# B&R Automation Studio project NAINV104C00R8L515F00 (part 31)

#### Act_Main.st
```iecst
(** 2019-04-08 **)
ACTION Act_Main:

	IF eStatOld <> eStat THEN
		fbFileOldDel1(bEn := FALSE);
		fbFileRead1(bEn := FALSE);
		fbFileWrite1(bEn := FALSE);

		sStatTxt	:= a_sStatText[eStat];

		eStatOld	:= eStat;

		eStatus		:= Busy;
	END_IF

	//Main
	CASE eStat OF

		HermesActIdle:
			eStatus	:= Idle;

		HermesActBGStartRun:
			IF eStatus = Idle OR eStatus = Busy THEN

				bRun	:= TRUE;
				bStop	:= FALSE;
				eStatus	:= Done;

			END_IF

		HermesActBGStopRun:
			IF eStatus = Idle OR eStatus = Busy THEN

				bStop	:= TRUE;
				eStatus	:= Done;

			END_IF

		HermesActDeleteOldLog:
			IF eStatus = Idle OR eStatus = Busy THEN

				eStatus	:= Busy;

				fbFileOldDel1.dtDTNow	:= p_dtCurrDT;
				fbFileOldDel1(bEn := TRUE);
				IF fbFileOldDel1.udiStatus = 0 THEN
					eStatus	:= Done;
				ELSIF fbFileOldDel1.udiStatus < 65534 THEN
					eStatus		:= Error;

					IF fbFileOldDel1.udiStatus = 1910 THEN
						udiStatus	:= 10111;	//Get Directory Info Error While Deleting Old Log
					ELSIF fbFileOldDel1.udiStatus = 1911 THEN
						udiStatus	:= 10112;	//Directory Read Error While Deleting Old Log
					ELSIF fbFileOldDel1.udiStatus = 1912 THEN
						udiStatus	:= 10113;	//File Delete Error While Deleting Old Log
					ELSE
						udiStatus	:= fbFileOldDel1.udiStatus;
					END_IF
				END_IF

			END_IF
		HermesActReadRetain:
			IF eStatus = Idle OR eStatus = Busy THEN

				eStatus	:= Busy;

				fbFileRead1(bEn := TRUE);

				IF fbFileRead1.udiStatus = 0 THEN
					eStatus	:= Done;

					a_tyBoardDepartedInfoWr := a_tyBoardDepartedInfo;
				ELSIF fbFileRead1.udiStatus < 65534 THEN
					eStatus	:= Error;

					IF fbFileRead1.udiStatus = 1900 THEN
						udiStatus	:= 10114;	//File Open Error While Reading Retain File
					ELSIF fbFileRead1.udiStatus = 1902 THEN
						udiStatus	:= 10115;	//File Read Error While Reading Retain File
					ELSIF fbFileRead1.udiStatus = 1904 THEN
						udiStatus	:= 10116;	//File Close Error While Reading Retain File
					ELSIF fbFileRead1.udiStatus = 1915 THEN
						eStatus			:= Done;
						bFileNotFound	:= TRUE;
					ELSE
						udiStatus	:= fbFileRead1.udiStatus;
					END_IF
				END_IF

			END_IF

		HermesActWriteRetain:
			IF eStatus = Idle OR eStatus = Busy THEN

				eStatus	:= Busy;

				fbFileWrite1(bEn := TRUE);

				IF fbFileWrite1.udiStatus = 0 THEN
					eStatus	:= Done;
				ELSIF fbFileWrite1.udiStatus < 65534 THEN
					eStatus	:= Error;

					IF fbFileWrite1.udiStatus = 1900 THEN
						udiStatus	:= 10117;	//File Open Error While Writing Retain File
					ELSIF fbFileWrite1.udiStatus = 1901 THEN
						udiStatus	:= 10118;	//File Create Error While Writing Retain File
					ELSIF fbFileWrite1.udiStatus = 1903 THEN
						udiStatus	:= 10119;	//File Write Error While Writing Retain File
					ELSIF fbFileWrite1.udiStatus = 1904 THEN
						udiStatus	:= 10120;	//File Close Error While Writing Retain File
					ELSIF fbFileWrite1.udiStatus = 1914 THEN
						udiStatus	:= 10121;	//Directory Does Not Exist While Writing Retain File
					ELSE
						udiStatus	:= fbFileWrite1.udiStatus;
					END_IF
				END_IF

			END_IF

		ELSE
			IF eStatus = Idle OR eStatus = Busy THEN
				eStatus	:= Done;
			END_IF

	END_CASE

END_ACTION
```

#### Init.st
```iecst
(** 2020-09-10 **)
PROGRAM _INIT

	(* Always Change If Project Change *)

	//Pass Address To Global Address For External Use
	//Action, State & Status
	p_DSHermes2Stat		:= ADR(eStat);
	p_DSHermes2Status	:= ADR(eMainStatus);
	p_DSHermes2StatTxt	:= ADR(sStatTxt);

	//Alarm
	p_DSHermes2AlmData	:= ADR(tyAlmData);
	p_DSHermes2AlmData1	:= ADR(tyAlmData1);
	p_DSHermes2AlmData2	:= ADR(tyAlmData2);
	p_DSHermes2AlmData3	:= ADR(tyAlmData3);
	p_DSHermes2AlmData4	:= ADR(tyAlmData4);

	//Output
	p_DSHermes2Connected			:= ADR(bConnected);
	p_DSHermes2HandshakeDone		:= ADR(bHandshakeDone);
	p_DSHermes2USRdy				:= ADR(bUSRdy);
	p_DSHermes2DSRdy				:= ADR(bDSRdy);
	p_DSHermes2USGdRdy				:= ADR(bUSGdRdy);
	p_DSHermes2DSGdRdy				:= ADR(bDSGdRdy);
	p_DSHermes2Transporting			:= ADR(bTransporting);
	p_DSHermes2StopTransport		:= ADR(bStopTransport);
	p_DSHermes2InternalSnd			:= ADR(sInternalSnd);

	p_DSHermes2TransportFinish		:=ADR(bTransportFinishedSnd);
	p_DSHermes2TransportFinishMsg	:= ADR(tyTransportFinished);
	//command
	p_DSHermes2CommandParam			:= ADR(tyCommandParam);
	//route
	p_DSHermes2BrdAvlSnd				:= ADR(tyBoardAvailableSnd);
	//p_DSHermes2RcvReverseUSMcRdy		:= ADR(bDSHermesRcvReverseUSMcRdy);
	(* Always Change If Project Change *)

END_PROGRAM
```

### RmtHermes.var - Change By Project
```iecst
(*2019-05-04*)
(**)
(*Action & State & Status*)
VAR
	p_RmtHermesStat : UDINT;
	p_RmtHermesStatus : UDINT;
	p_RmtHermesStatTxt : UDINT;
	p_RmtHermesAct : UDINT;
	p_RmtHermesMcParamAct : UDINT;
END_VAR
(**)
(*Alarm*)
VAR
	p_RmtHermesAlmData : UDINT;
	p_RmtHermesAlmData1 : UDINT;
	p_RmtHermesAlmData2 : UDINT;
	p_RmtHermesAlmData3 : UDINT;
	p_RmtHermesInfoData : UDINT;
END_VAR
(**)
(*Output*)
VAR
	p_RmtHermesFileNotFound : UDINT;
	p_RmtHermesConnected : UDINT;
	p_RmtHermesWriteConfig : UDINT;
	p_RmtHermesUpdateUIData : UDINT;
	p_RmtHermesSetConfiguration : UDINT;
	p_RmtHermesFoundIndexUS1 : UDINT;
	p_RmtHermesFoundIndexUS2 : UDINT;
	p_RmtHermesFoundIndexUS3 : UDINT;
	p_RmtHermesFoundIndexUS4 : UDINT;
	p_RmtHermesFoundIndexDS1 : UDINT;
	p_RmtHermesFoundIndexDS2 : UDINT;
	p_RmtHermesFoundIndexDS3 : UDINT;
	p_RmtHermesFoundIndexDS4 : UDINT;
	p_RmtHermesIndexUS1 : UDINT;
	p_RmtHermesIndexUS2 : UDINT;
	p_RmtHermesIndexUS3 : UDINT;
	p_RmtHermesIndexUS4 : UDINT;
	p_RmtHermesIndexDS1 : UDINT;
	p_RmtHermesIndexDS2 : UDINT;
	p_RmtHermesIndexDS3 : UDINT;
	p_RmtHermesIndexDS4 : UDINT;
	p_RmtHermesCurrentConfiguration : UDINT;
	p_RmtHermesCurrentConfMcId : UDINT;
END_VAR
```

### Program Logical/Hermes/RmtHermes (IEC, version 1.00.0) - 1.00.0 - NtHermes v5.00.0 , NtTCP v5.00.0 , NtMessage v5.00.0

#### Init.st - Change By Project
```iecst
(** 2021-08-01 **)
PROGRAM _INIT

	(* Always Change If Project Change *)

	//Pass Address To Global Address For External Use
	//Action, State & Status
	p_RmtHermesStat	    	:= ADR(eStat);
	p_RmtHermesStatus   	:= ADR(eMainStatus);
	p_RmtHermesStatTxt   	:= ADR(sStatTxt);
	p_RmtHermesAct	    	:= ADR(eHermesAct);
	p_RmtHermesMcParamAct	:= ADR(eMcParamAct);

	//Alarm
	p_RmtHermesAlmData	    := ADR(tyAlmData);
	p_RmtHermesAlmData1	    := ADR(tyAlmData1);
	p_RmtHermesAlmData2	    := ADR(tyAlmData2);
	p_RmtHermesAlmData3	    := ADR(tyAlmData3);
	p_RmtHermesInfoData	    := ADR(tyInfoData);

	//Output
	p_RmtHermesFileNotFound			:= ADR(bFileNotFound);
	p_RmtHermesConnected			:= ADR(bConnected);
	p_RmtHermesSetConfiguration	    := ADR(tySetConfiguration);
	p_RmtHermesWriteConfig          := ADR(bWriteConfig);
	p_RmtHermesUpdateUIData	        := ADR(bUpdateUIData);

	//Data
	p_RmtHermesFoundIndexUS1              := ADR(bFoundIndexUS1);
	p_RmtHermesFoundIndexUS2              := ADR(bFoundIndexUS2);
	p_RmtHermesFoundIndexUS3              := ADR(bFoundIndexUS3);
	p_RmtHermesFoundIndexUS4              := ADR(bFoundIndexUS4);
	p_RmtHermesFoundIndexDS1              := ADR(bFoundIndexDS1);
	p_RmtHermesFoundIndexDS2              := ADR(bFoundIndexDS2);
	p_RmtHermesFoundIndexDS3              := ADR(bFoundIndexDS3);
	p_RmtHermesFoundIndexDS4              := ADR(bFoundIndexDS4);
	p_RmtHermesIndexUS1                   := ADR(udiFoundIndexUS1);
	p_RmtHermesIndexUS2                   := ADR(udiFoundIndexUS2);
	p_RmtHermesIndexUS3                   := ADR(udiFoundIndexUS3);
	p_RmtHermesIndexUS4                   := ADR(udiFoundIndexUS4);
	p_RmtHermesIndexDS1                   := ADR(udiFoundIndexDS1);
	p_RmtHermesIndexDS2                   := ADR(udiFoundIndexDS2);
	p_RmtHermesIndexDS3                   := ADR(udiFoundIndexDS3);
	p_RmtHermesIndexDS4                   := ADR(udiFoundIndexDS4);
//	p_RmtHermesCurrentConfiguration	:= ADR(tyCurrentConfiguration);
//	p_RmtHermesCurrentConfMcId		:= ADR(tyCurrentConfiguration.tyData.sMachineId);

	(* Always Change If Project Change *)
END_PROGRAM
```

#### Act_InitGlobal.st - Change By Project
```iecst
(** 2021-08-01 **)
ACTION Act_InitGlobal:

	(* Always Change If Project Change *)

	//Pass Data To Link
	p_bLinkStartupRun ACCESS p_StartupRun;

	//Pass Data To Internal Use
	p_udiRstErr ACCESS p_RstErrReset;
	p_bPrep ACCESS p_NtParamHermesPrep;
	p_sIPAddr ACCESS p_HWInfoIPAddr;
	p_tyDTStructure ACCESS p_TimeCurrDTStruct;
	p_dtCurrDT ACCESS p_TimeCurrDT;
	p_sMcId ACCESS p_McParamMcNm;
	p_bRmtPrep ACCESS p_NtParamHermesRmtPrep;
	p_bRmtEn ACCESS p_McParamHermesRmtEn;
	p_udiSndBffrSize ACCESS p_NtParamRmtHermesSndBffrSize;
	p_udiRcvBffrSize ACCESS p_NtParamRmtHermesRcvBffrSize;
	p_udiAliveIdleTimeInSec ACCESS p_NtParamRmtHermesAliveTmInSec;
	p_udiFileKeepDay ACCESS p_NtParamRmtHermesFileKeepDay;
	p_sConfigFileName ACCESS p_NtParamRmtHermesConfigFileNm;
	p_sProgNm ACCESS p_NtParamRmtHermesProgNm;
	p_bNtSettingsLoadDone ACCESS p_StartupNtSettingsLoadDone;
	p_tyHermesConfiguration ACCESS p_HermesConfiguration;
	p_eHermesStat ACCESS p_HermesStat;
	p_eHermesStatus ACCESS p_HermesStatus;
	p_eMcParamStat ACCESS p_McParamStat;
	p_eMcParamStatus ACCESS p_McParamStatus;
	p_iInput ACCESS p_NtParamHermesInput;
	p_iOutput ACCESS p_NtParamHermesOutput;

	(* Always Change If Project Change *)
END_ACTION
```

#### InputRef_Link.var - Change By Project
```iecst
(*2021-08-01*)
(**)
VAR
	p_bLinkStartupRun : REFERENCE TO BOOL;
	bRmtHermesRun : BOOL;
	bRmtHermesStop : BOOL;
END_VAR
```

#### Act_LinkAction.st - Change By Project
```iecst
(** 2021-08-01 **)
ACTION Act_LinkAction:

	IF p_bLinkStartupRun = TRUE THEN
		p_eAct ACCESS p_StartupRmtHermesAct;
	ELSE
		p_eAct ACCESS ADR(eAct);

		IF EDGEPOS(p_bRmtPrep AND p_bRmtEn) THEN
			bRmtHermesRun	:= TRUE;
			bRmtHermesStop	:= FALSE;
		END_IF

		IF EDGENEG(p_bRmtPrep) OR EDGENEG(p_bRmtEn) THEN
			bRmtHermesRun	:= FALSE;
			bRmtHermesStop	:= TRUE;
		END_IF

		IF bRmtHermesRun = TRUE THEN
			p_eAct	:= HermesActBGStartRun;

			IF (eStat = HermesActBGStartRun) AND (eStatus = Done) THEN
				p_eAct			:= HermesActIdle;
				bRmtHermesRun	:= FALSE;
			END_IF
		END_IF

		IF bRmtHermesStop = TRUE THEN
			p_eAct	:= HermesActBGStopRun;

			IF (eStat = HermesActBGStopRun) AND (eStatus = Done) THEN
				p_eAct			:= HermesActIdle;
				bRmtHermesStop	:= FALSE;
			END_IF
		END_IF

	END_IF

END_ACTION
```

#### Act_LinkEn.st - Change By Project
```iecst
(** 2021-08-01 **)
ACTION Act_LinkEn:

	//Link bPrep, bEn & bDis

END_ACTION
```

#### Act_Link.st - Change By Project
```iecst
(** 2021-08-01 **)
ACTION Act_Link:

	//Info Message
	p_sInfoMsg		:= 'Hermes Configuration Received From Remote Station';

	IF	p_iInput > (DINT_TO_INT(c_diHermesConfigMaxIdx)+1) THEN
		p_iInput := (DINT_TO_INT(c_diHermesConfigMaxIdx)+1); //capped at limit
	END_IF

	IF	p_iOutput > (DINT_TO_INT(c_diHermesConfigMaxIdx)+1) THEN
		p_iOutput := (DINT_TO_INT(c_diHermesConfigMaxIdx)+1); //capped at limit
	END_IF

END_ACTION
```

#### Cyclic.st - Do Not Change!!!
```iecst
(** 2021-08-01 **)
PROGRAM _CYCLIC

	IF bInitDone = FALSE THEN
		bInitDone	:= TRUE;

		Act_InitLocal;
		Act_InitGlobal;

	ELSIF bInitialDone = FALSE THEN
		IF p_bNtSettingsLoadDone = TRUE THEN
			bInitialDone	:= TRUE;

			Act_Initial;
		END_IF

	ELSE

		Act_RstErr;
		Act_LinkAction;
		Act_Action;
		Act_LinkEn;

		IF (p_bPrep = TRUE) AND (p_bEn = TRUE) AND (p_bDis = FALSE) THEN
			Act_Link;
			Act_Main;
			Act_Background;
			Act_Background_ProcessData;
		ELSE
			Act_Main_Disable;

			IF eStat <> HermesActIdle THEN
				eStatus	:= Done;
			ELSE
				eStatus	:= Idle;
			END_IF
		END_IF

		Act_CombineErr;
		Act_Alarm;
		Act_Alarm1;
		Act_Alarm2;
		Act_Alarm3;

	END_IF

END_PROGRAM
```

#### Act_RstErr.st - Do Not Change!!!
```iecst
(** 2021-08-01 **)
ACTION Act_RstErr:

	IF p_udiRstErr <> udiRstErrOld THEN
		bRstErr			:= TRUE;
		udiRstErrOld	:= p_udiRstErr;
	ELSE
		bRstErr			:= FALSE;
	END_IF

END_ACTION
```

#### Act_InitLocal.st - Do Not Change!!!
```iecst
(** 2021-08-01 **)
ACTION Act_InitLocal:

	//Input Reference Link To Local Variable
	p_eAct ACCESS ADR(eAct);
	p_udiRstErr ACCESS ADR(udiRstErr);
	p_bPrep ACCESS ADR(bPrep);
	p_bEn ACCESS ADR(bEn);
	p_bDis ACCESS ADR(bDis);
	p_tyParam ACCESS ADR(tyParam);
	p_sIPAddr ACCESS ADR(sIPAddr);
	p_tyDTStructure ACCESS ADR(tyDTStructure);
	p_dtCurrDT ACCESS ADR(dtCurrDT);
	p_sMcId ACCESS ADR(sMcId);
	p_bRmtPrep ACCESS ADR(bRmtPrep);
	p_bRmtEn ACCESS ADR(bRmtEn);
	p_udiSndBffrSize ACCESS ADR(udiSndBffrSize);
	p_udiRcvBffrSize ACCESS ADR(udiRcvBffrSize);
	p_udiAliveIdleTimeInSec ACCESS ADR(udiAliveIdleTimeInSec);
	p_udiFileKeepDay ACCESS ADR(udiFileKeepDay);
	p_sConfigFileName ACCESS ADR(sConfigFileName);
	p_sProgNm ACCESS ADR(sProgNm);
	p_bNtSettingsLoadDone ACCESS ADR(bNtSettingsLoadDone);
	p_sInfoMsg ACCESS ADR(sInfoMsg);
	p_bNtSettingsLoadDone ACCESS ADR(bNtSettingsLoadDone);
	p_sInfoMsg ACCESS ADR(sInfoMsg);
	p_tyHermesConfiguration ACCESS ADR(tyHermesCurrConfiguration);
	p_iInput ACCESS ADR(iInput);
	p_iOutput ACCESS ADR(iOutput);

END_ACTION
```

#### Act_Initial.st - Do Not Change!!!
```iecst
(** 2021-08-01 **)
ACTION Act_Initial:

	//Initial
	sStatTxt	:= a_sStatText[eStat];

	fbCreateSvr.udiSndBffrSize		:= p_udiSndBffrSize;
	fbCreateSvr.udiRcvBffrSize		:= p_udiRcvBffrSize;
	fbCreateSvr.udiAliveIdleTmInSec	:= p_udiAliveIdleTimeInSec;
	fbCreateSvr(bEn := FALSE);

	fbListen(bEn := FALSE);

	fbRcv.udiBffrSize	:= SIZEOF(sRcv);
	fbRcv.p_BffrDest	:= ADR(sRcv);
	fbRcv(bEn := FALSE);

	fbSend.p_BffrDest	:= ADR(sSnd);
	fbSend(bEn := FALSE);

	fbCloseSvr(bEn := FALSE);
	fbCloseClnt(bEn := FALSE);

	fbParseXMLTable.p_XMLTable	:= ADR(a_tyXMLTableDataRcv);

	fbFileAppend1.sDevice	:= 'Log';
	fbFileAppend1(bEn := FALSE);

	fbFileOldDel1.sDevice			:= 'Log';
	fbFileOldDel1.sPath				:= '';
	fbFileOldDel1.sKeyword			:= p_sProgNm;
	fbFileOldDel1.udiFileKeepDay	:= p_udiFileKeepDay;
	fbFileOldDel1(bEn := FALSE);

END_ACTION
```

#### Act_Action.st - Do Not Change!!!
```iecst
(** 2021-08-01 **)
ACTION Act_Action:

	//Reset Error
	IF (eStatus = Error) AND bRstErr THEN
		p_eAct	:= HermesActIdle;
		eStat	:= HermesActIdle;
	END_IF

	//Set p_eAct
	IF eStatus = Idle OR eStatus = Busy OR eStatus = Done THEN
		eStat	:= p_eAct;
	END_IF

END_ACTION
```

#### Act_Main.st - Do Not Change!!!
```iecst
(** 2021-08-01 **)
ACTION Act_Main:

	IF eStatOld <> eStat THEN
		fbFileOldDel1(bEn := FALSE);
		bFileNotFound	:= FALSE;
		sStatTxt	:= a_sStatText[eStat];

		eStatOld	:= eStat;

		eStatus		:= Busy;
	END_IF

	//Main
	CASE eStat OF

		HermesActIdle:
			eStatus	:= Idle;

		HermesActBGStartRun:
			IF eStatus = Idle OR eStatus = Busy THEN

				bRun	:= TRUE;
				bStop	:= FALSE;
				eStatus	:= Done;

			END_IF

		HermesActBGStopRun:
			IF eStatus = Idle OR eStatus = Busy THEN

				bStop	:= TRUE;
				eStatus	:= Done;

			END_IF

		HermesActDeleteOldLog:
			IF eStatus = Idle OR eStatus = Busy THEN

				eStatus	:= Busy;

				fbFileOldDel1.dtDTNow	:= p_dtCurrDT;
				fbFileOldDel1(bEn := TRUE);
				IF fbFileOldDel1.udiStatus = 0 THEN
					eStatus	:= Done;
				ELSIF fbFileOldDel1.udiStatus < 65534 THEN
					eStatus		:= Error;

					IF fbFileOldDel1.udiStatus = 1910 THEN
						udiStatus	:= 10111;	//Get Directory Info Error While Deleting Old Log
					ELSIF fbFileOldDel1.udiStatus = 1911 THEN
						udiStatus	:= 10112;	//Directory Read Error While Deleting Old Log
					ELSIF fbFileOldDel1.udiStatus = 1912 THEN
						udiStatus	:= 10113;	//File Delete Error While Deleting Old Log
					ELSE
						udiStatus	:= fbFileOldDel1.udiStatus;
					END_IF
				END_IF

			END_IF

		ELSE
			IF eStatus = Idle OR eStatus = Busy THEN
				eStatus	:= Done;
			END_IF

	END_CASE

END_ACTION
```

#### Act_Background.st - Do Not Change!!!
```iecst
(** 2021-08-01 **)
ACTION Act_Background:

	IF bRun = TRUE THEN
		IF udiSvrIdent = 0 THEN
			Act_Background_TCPCreateSvr;

			tyParamOld	:= p_tyParam;

		ELSE
			IF bRstConnection = FALSE THEN

				IF udiClntIdent = 0 THEN
					Act_Background_TCPListen;
				END_IF

				IF udiClntIdent <> 0 THEN
					Act_Background_TCPRcv;
				END_IF

				Act_Background_NotificationRcv;

				Act_Background_IllegalMsg;
				Act_Background_UpdtConfig;

				Act_Background_SendConfig;

				Act_Background_Err;

				IF udiClntIdent <> 0 THEN
					Act_Background_TCPSend;
				END_IF

				Act_Background_Log;

			ELSE
				IF udiClntIdent <> 0 THEN
					Act_Background_TCPCloseClnt;
				ELSE
					IF udiSvrIdent <> 0 THEN
						Act_Background_TCPCloseSvr;
					END_IF
				END_IF

			END_IF

		END_IF

		Act_Background_Stop;

	END_IF

	IF EDGENEG(bRun) OR EDGENEG(udiSvrIdent = 0) THEN
		//Reset
		fbCreateSvr(bEn := FALSE);
	END_IF

	IF EDGENEG(bRun) OR EDGENEG(udiClntIdent = 0) THEN
		//Reset
		fbListen(bEn := FALSE);

		bConnected	:= bRun;
	END_IF

	IF EDGENEG(bRun) OR EDGENEG(udiSvrIdent <> 0) OR EDGENEG(udiClntIdent <> 0) THEN
		fbRcv(bEn := FALSE);
		fbSend(bEn := FALSE);

		bConnected		:= FALSE;

		memset(ADR(a_eMsgSend) , 0 , SIZEOF(a_eMsgSend));
		udiMsgSendBffr	:= 0;
	END_IF

	IF EDGENEG(bRun) THEN
		fbFileAppend1(bEn := FALSE);
		iWriteLogStep	:= 0;

		memset(ADR(tyMsgTypeRcv) , 0 , SIZEOF(tyMsgTypeRcv));
	END_IF

	IF EDGENEG(bRun) OR EDGENEG(udiSvrIdent <> 0) THEN
		bRstConnection	:= FALSE;
		fbCloseSvr(bEn := FALSE);
	END_IF

	IF EDGENEG(bRun) OR EDGENEG(udiClntIdent <> 0) THEN
		fbCloseClnt(bEn := FALSE);
	END_IF

	//Reset Error
	IF (eStatus1 = Error) AND bRstErr THEN
		eStatus1	:= Idle;
		udiStatus1	:= 0;

		fbCreateSvr(bEn := FALSE);
		fbListen(bEn := FALSE);
		fbRcv(bEn := FALSE);
		fbSend(bEn := FALSE);
		fbCloseSvr(bEn := FALSE);
		fbCloseClnt(bEn := FALSE);

		fbFileAppend1(bEn := FALSE);
		iWriteLogStep	:= 0;

		bConnected		:= FALSE;
		bRstConnection	:= FALSE;

		memset(ADR(tyMsgTypeRcv) , 0 , SIZEOF(tyMsgTypeRcv));
		memset(ADR(a_eMsgSend) , 0 , SIZEOF(a_eMsgSend));
		udiMsgSendBffr	:= 0;
	END_IF

	IF (eStatus2 = Error) AND bRstErr THEN
		eStatus2	:= Idle;
		udiStatus2	:= 0;

	END_IF

	IF (eStatus3 = Error) AND bRstErr THEN
		eStatus3	:= Idle;
		udiStatus3	:= 0;

		fbFileAppend1(bEn := FALSE);
		iWriteLogStep	:= 0;
	END_IF

END_ACTION
```

#### Act_Background_ProcessData.st - Do Not Change!!!
```iecst
(** 2021-08-01 **)
ACTION Act_Background_ProcessData:

	//Write Config into "Hermes"
	fbDelayTm(IN := bWriteConfig, PT := T#0.5S); //Delay 0.5s to let Hermes take the Data, before WriteConfig

	IF fbDelayTm.Q THEN

		eHermesAct := HermesActWriteConfig;
		eMcParamAct := McParamActWrite;

		IF p_eHermesStatus = Done AND p_eHermesStat = HermesActWriteConfig AND p_eMcParamStat = McParamActWrite AND p_eMcParamStatus = Done THEN

			eMcParamAct     := McParamActIdle;
			eHermesAct		:= HermesActIdle;
			bWriteConfig    := FALSE;
			bUpdateUIData   := TRUE;
			fbDelayTm(IN := FALSE);
			tyInfoData.sProgNm		:= p_sProgNm;
			tyInfoData.udiCode		:= 10000;
			tyInfoData.eSeverity	:= AlmSeverityInfo;
			tyInfoData.sAlmMsg		:= p_sInfoMsg;

		ELSIF  (p_eHermesStatus = Error AND p_eHermesStat = HermesActWriteConfig) OR (p_eMcParamStat = McParamActWrite AND p_eMcParamStatus = Error)  THEN

			eMcParamAct     := McParamActIdle;
			eHermesAct		:= HermesActIdle;
			bWriteConfig    := FALSE;
			bUpdateUIData   := FALSE;
			fbDelayTm(IN := FALSE);

			fHermesAddOneMsgSend(ADR(a_eMsgSend) , ADR(udiMsgSendBffr) , HermesMsgTypeNotification);

			udiStatus2 := 10199; //SetConfiguration Failed, Please Send Again Or Set in Machine HMI back
			tyNotificationSnd.tyAvl.bSeverity			:= TRUE;
			tyNotificationSnd.tyAvl.bNotificationCode	:= TRUE;
			tyNotificationSnd.tyAvl.bDescription		:= TRUE;
			tyNotificationSnd.tyData.eSeverity			:= HermesSeverityFatalError;
			tyNotificationSnd.tyData.iNotificationCode	:= UDINT_TO_INT(udiStatus2);
			tyNotificationSnd.tyData.sDescription		:= a_tyAlmText[udiStatus2].sAlmText;

		END_IF
	END_IF

	//Update UI
	IF bUpdateUIData THEN
		tyInfoData.sProgNm		:= p_sProgNm;
		tyInfoData.udiCode		:= 10000;
		tyInfoData.eSeverity	:= AlmSeverityInfo;
		tyInfoData.sAlmMsg		:= p_sInfoMsg;
	END_IF

	//Auto Reset Info Pop Up
	fbDelayTm1(IN := bUpdateUIData , PT := T#2S); //Auto reset at the Moment (Can Be Changed if need)
	IF fbDelayTm1.Q = TRUE THEN

		//Clear Info Message
		tyInfoData.sProgNm		:= '';
		tyInfoData.udiCode		:= 0;
		tyInfoData.eSeverity	:= AlmSeverityNA;
		tyInfoData.sAlmMsg		:= '';

		bUpdateUIData := FALSE;
		bFoundIndexUS1 := FALSE;
		bFoundIndexUS2 := FALSE;
		bFoundIndexUS3 := FALSE;
		bFoundIndexUS4 := FALSE;
		bFoundIndexDS1 := FALSE;
		bFoundIndexDS2 := FALSE;
		bFoundIndexDS3 := FALSE;
		bFoundIndexDS4 := FALSE;
		fbDelayTm1(IN := FALSE);
	END_IF

END_ACTION
```

#### Act_Background_TCPCreateSvr.st - Do Not Change!!!
```iecst
(** 2021-08-01 **)
ACTION Act_Background_TCPCreateSvr:

	IF eStatus1 <> Error THEN

		//Create Server
		fbCreateSvr.sSvrIP				:= p_sIPAddr;
		fbCreateSvr.uiSvrPort			:= p_tyParam.uiSvrPort; //default = 1248
		fbCreateSvr(bEn := TRUE);

		IF fbCreateSvr.udiStatus = 0 THEN
			udiSvrIdent	:= fbCreateSvr.udiTCPIdent;
			fbCreateSvr(bEn := FALSE);

		ELSIF fbCreateSvr.udiStatus < 65534 THEN
			eStatus1	:= Error;

			IF fbCreateSvr.udiStatus = 2300 THEN
				udiStatus1	:= 10000;	//Invalid Ident While Creating Server
			ELSIF fbCreateSvr.udiStatus = 2302 THEN
				udiStatus1	:= 10001;	//Setting Keep Alive Interval Time Error While Creating Server
			ELSIF fbCreateSvr.udiStatus = 2303 THEN
				udiStatus1	:= 10002;	//Setting Keep Alive Idle Time Error While Creating Server
			ELSIF fbCreateSvr.udiStatus = 2304 THEN
				udiStatus1	:= 10003;	//Setting Keep Alive Count Error While Creating Server
			ELSIF fbCreateSvr.udiStatus = 2305 THEN
				udiStatus1	:= 10004;	//Setting Keep Alive Error While Creating Server
			ELSIF fbCreateSvr.udiStatus = 2306 THEN
				udiStatus1	:= 10005;	//Setting Receive Buffer Error While Creating Server
			ELSIF fbCreateSvr.udiStatus = 2307 THEN
				udiStatus1	:= 10006;	//Setting Send Buffer Error While Creating Server
			ELSIF fbCreateSvr.udiStatus = 2308 THEN
				udiStatus1	:= 10007;	//Setting No Waiting Error While Creating Server
			ELSIF fbCreateSvr.udiStatus = 2309 THEN
				udiStatus1	:= 10008;	//TCP Open Port Error While Creating Server
			ELSIF fbCreateSvr.udiStatus = 2310 THEN
				udiStatus1	:= 10009;	//Closing TCP Error While Creating Server
			ELSE
				udiStatus1	:= fbCreateSvr.udiStatus;
			END_IF

		END_IF

	END_IF

END_ACTION
```

#### Act_Background_TCPListen.st - Do Not Change!!!
```iecst
(** 2021-08-01 **)
ACTION Act_Background_TCPListen:

	IF eStatus1 <> Error AND eStatus2 <> Error THEN

		fbListen.udiSvrIdent	:= udiSvrIdent;
		fbListen(bEn := TRUE);

		IF fbListen.udiStatus = 0 THEN
			udiClntIdent	:= fbListen.udiClntIdent;
			fbListen(bEn := FALSE);

		ELSIF fbListen.udiStatus = 2311 THEN
			fbListen(bEn := FALSE);

		ELSIF fbListen.udiStatus < 65534 THEN
			eStatus1	:= Error;

			IF fbListen.udiStatus = 2300 THEN
				udiStatus1	:= 10010;	//Invalid Ident While Listening Client
			ELSIF fbListen.udiStatus = 2312 THEN
				udiStatus1	:= 10012;	//Listen To Client Error While Listening Client
			ELSE
				udiStatus1	:= fbListen.udiStatus;
			END_IF

		END_IF

	END_IF

END_ACTION
```

#### Act_Background_TCPRcv.st - Do Not Change!!!
```iecst
(** 2021-08-01 **)
ACTION Act_Background_TCPRcv:

	IF eStatus1 <> Error THEN

		//Receive Data
		fbRcv.udiTCPIdent	:= udiClntIdent;
		fbRcv(bEn := TRUE);

		IF fbRcv.udiStatus = 0 THEN

			fLogDTConvert(ADR(sDT) , p_dtCurrDT);
			memset(ADR(a_sLogList[udiLogCntr]) , 0 , SIZEOF(a_sLogList[udiLogCntr]));
			memcpy(ADR(a_sLogList[udiLogCntr]) + LEN(a_sLogList[udiLogCntr]) , ADR(sDT) , LEN(sDT));
			memcpy(ADR(a_sLogList[udiLogCntr]) + LEN(a_sLogList[udiLogCntr]) , ADR('$r$n') , LEN('$r$n'));
			memcpy(ADR(a_sLogList[udiLogCntr]) + LEN(a_sLogList[udiLogCntr]) , ADR('RCV_FRM_RMT$r$n') , LEN('RCV_FRM_RMT$r$n'));
			memcpy(ADR(a_sLogList[udiLogCntr]) + LEN(a_sLogList[udiLogCntr]) , ADR(sRcv) , LEN(sRcv));
			memcpy(ADR(a_sLogList[udiLogCntr]) + LEN(a_sLogList[udiLogCntr]) , ADR('$r$n$r$n') , LEN('$r$n$r$n'));

			udiLogCntr	:= udiLogCntr + 1;
			IF udiLogCntr = 11 THEN
				udiLogCntr	:= 1;
			END_IF

			fXMLConvertToTable(ADR(sRcv) , LEN(sRcv) , ADR(a_tyXMLTableDataRcv) , ADR(a_tyXMLTableDataRcv[0].sTitle) , SIZEOF(a_tyXMLTableDataRcv[0].sTitle) , ADR(a_tyXMLTableDataRcv[0].sValue) , SIZEOF(a_tyXMLTableDataRcv[0].sValue) , ADR(a_tyXMLTableDataRcv[0].uiSize) , SIZEOF(a_tyXMLTableDataRcv[0]) , SIZEOF(a_tyXMLTableDataRcv) / SIZEOF(a_tyXMLTableDataRcv[0]) , ADR(udiXMLTableWriteIdx));

			fbParseXMLTable.iTotalIdxWrite	:= UDINT_TO_INT(udiXMLTableWriteIdx);
			fbParseXMLTable;

			IF fbParseXMLTable.tyMsgType.bCheckAlive = TRUE THEN
				tyMsgTypeRcv.bCheckAlive	:= TRUE;
				tyCheckAlive				:= fbParseXMLTable.tyCheckAlive;
			END_IF

			IF fbParseXMLTable.tyMsgType.bCheckAlivePing = TRUE THEN
				tyMsgTypeRcv.bCheckAlivePing	:= TRUE;
				tyCheckAlivePing				:= fbParseXMLTable.tyCheckAlivePing;
			END_IF

			IF fbParseXMLTable.tyMsgType.bCheckAlivePong = TRUE THEN
				tyMsgTypeRcv.bCheckAlivePong	:= TRUE;
				tyCheckAlivePong				:= fbParseXMLTable.tyCheckAlivePong;
			END_IF

			IF fbParseXMLTable.tyMsgType.bServiceDescription = TRUE THEN
				tyMsgTypeRcv.bServiceDescription	:= TRUE;
				tyServiceDescriptionRcv				:= fbParseXMLTable.tyServiceDescription;
			END_IF

			IF fbParseXMLTable.tyMsgType.bNotification = TRUE THEN
				tyMsgTypeRcv.bNotification	:= TRUE;
				tyNotificationRcv			:= fbParseXMLTable.tyNotification;
			END_IF

			IF fbParseXMLTable.tyMsgType.bBoardAvailable = TRUE THEN
				tyMsgTypeRcv.bBoardAvailable	:= TRUE;
				tyBoardAvailableRcv				:= fbParseXMLTable.tyBoardAvailable;

			END_IF

			IF fbParseXMLTable.tyMsgType.bRevokeBoardAvailable = TRUE THEN
				tyMsgTypeRcv.bRevokeBoardAvailable	:= TRUE;
			END_IF

			IF fbParseXMLTable.tyMsgType.bMachineReady = TRUE THEN
				tyMsgTypeRcv.bMachineReady	:= TRUE;
				tyMachineReady				:= fbParseXMLTable.tyMachineReady;
			END_IF

			IF fbParseXMLTable.tyMsgType.bRevokeMachineReady = TRUE THEN
				tyMsgTypeRcv.bRevokeMachineReady	:= TRUE;
			END_IF

			IF fbParseXMLTable.tyMsgType.bStartTransport = TRUE THEN
				tyMsgTypeRcv.bStartTransport	:= TRUE;
				tyStartTransport				:= fbParseXMLTable.tyStartTransport;
			END_IF

			IF fbParseXMLTable.tyMsgType.bStopTransport = TRUE THEN
				tyMsgTypeRcv.bStopTransport	:= TRUE;
				tyStopTransport				:= fbParseXMLTable.tyStopTransport;
			END_IF

			IF fbParseXMLTable.tyMsgType.bTransportFinished = TRUE THEN
				tyMsgTypeRcv.bTransportFinished	:= TRUE;
				tyTransportFinished				:= fbParseXMLTable.tyTransportFinished;
			END_IF

			IF fbParseXMLTable.tyMsgType.bSetConfiguration = TRUE THEN
				tyMsgTypeRcv.bSetConfiguration	:= TRUE;
				tySetConfigurationRcv			:= fbParseXMLTable.tySetConfiguration;
			END_IF

			IF fbParseXMLTable.tyMsgType.bGetConfiguration = TRUE THEN
				tyMsgTypeRcv.bGetConfiguration	:= TRUE;
			END_IF

			IF fbParseXMLTable.tyMsgType.bCurrentConfiguration = TRUE THEN
				tyMsgTypeRcv.bCurrentConfiguration	:= TRUE;
				tyCurrentConfigurationRcv			:= fbParseXMLTable.tyCurrentConfiguration;
			END_IF

			IF fbParseXMLTable.tyMsgType.bBoardForecast = TRUE THEN
				tyMsgTypeRcv.bBoardForecast	:= TRUE;
				tyBoardForecast				:= fbParseXMLTable.tyBoardForecast;
			END_IF

			IF fbParseXMLTable.tyMsgType.bQueryBoardInfo = TRUE THEN
				tyMsgTypeRcv.bQueryBoardInfo	:= TRUE;
				tyQueryBoardInfo				:= fbParseXMLTable.tyQueryBoardInfo;
			END_IF

			IF fbParseXMLTable.tyMsgType.bSendBoardInfo = TRUE THEN
				tyMsgTypeRcv.bSendBoardInfo	:= TRUE;
				tySendBoardInfo				:= fbParseXMLTable.tySendBoardInfo;
			END_IF

			fbRcv(bEn := FALSE);

			memset(ADR(sRcv) , 0 , SIZEOF(sRcv));

		ELSIF fbRcv.udiStatus = 2317 THEN
			fbRcv(bEn := FALSE);

			memset(ADR(sRcv) , 0 , SIZEOF(sRcv));

		ELSIF fbRcv.udiStatus = 2316 THEN
			bRstConnection	:= TRUE;

			memset(ADR(sRcv) , 0 , SIZEOF(sRcv));

		ELSIF fbRcv.udiStatus = 2318 THEN
			bRstConnection	:= TRUE;

			memset(ADR(sRcv) , 0 , SIZEOF(sRcv));

		ELSIF fbRcv.udiStatus < 65534 THEN
			eStatus1	:= Error;

			IF fbRcv.udiStatus = 2300 THEN
				udiStatus1	:= 10014;	//Invalid Ident While Receiving Data
			ELSIF fbRcv.udiStatus = 2319 THEN
				udiStatus1	:= 10015;	//TCP Receive Data Error While Receiving Data
			ELSE
				udiStatus1	:= fbRcv.udiStatus;
			END_IF

			memset(ADR(sRcv) , 0 , SIZEOF(sRcv));

		END_IF

	END_IF

END_ACTION
```

#### Act_Background_NotificationRcv.st - Do Not Change!!!
```iecst
(** 2021-08-01 **)
ACTION Act_Background_NotificationRcv:

	IF eStatus1 <> Error THEN

		IF tyMsgTypeRcv.bNotification = TRUE THEN
			tyMsgTypeRcv.bNotification	:= FALSE;

			bRstConnection	:= fHermesNotificationRstConn(tyNotificationRcv) OR bRstConnection;

		END_IF

	END_IF

END_ACTION
```

#### Act_Background_IllegalMsg.st - Do Not Change!!!
```iecst
(** 2021-08-01 **)
ACTION Act_Background_IllegalMsg:

	IF eStatus2 <> Error THEN

		udiStatus2	:= fHermesIllegalMsgRmt(tyMsgTypeRcv);

		IF udiStatus2 <> 0 THEN
			eStatus2	:= Error;

			IF udiStatus2 = 2925 THEN
				udiStatus2	:= 10114;	//Receive Check Alive While In Remote Configuration
			ELSIF udiStatus2 = 2926 THEN
				udiStatus2	:= 10115;	//Receive Check Alive Ping While In Remote Configuration
			ELSIF udiStatus2 = 2927 THEN
				udiStatus2	:= 10116;	//Receive Check Alive Pong While In Remote Configuration
			ELSIF udiStatus2 = 2928 THEN
				udiStatus2	:= 10117;	//Receive ServiceDescription While In Remote Configuration
			ELSIF udiStatus2 = 2929 THEN
				udiStatus2	:= 10118;	//Receive BoardAvailable While In Remote Configuration
			ELSIF udiStatus2 = 2930 THEN
				udiStatus2	:= 10119;	//Receive RevokeBoardAvailable While In Remote Configuration
			ELSIF udiStatus2 = 2931 THEN
				udiStatus2	:= 10120;	//Receive MachineReady While In Remote Configuration
			ELSIF udiStatus2 = 2932 THEN
				udiStatus2	:= 10121;	//Receive RevokeMachineReady While In Remote Configuration
			ELSIF udiStatus2 = 2933 THEN
				udiStatus2	:= 10122;	//Receive StartTransport While In Remote Configuration
			ELSIF udiStatus2 = 2934 THEN
				udiStatus2	:= 10123;	//Receive StopTransport While In Remote Configuration
			ELSIF udiStatus2 = 2935 THEN
				udiStatus2	:= 10124;	//Receive TransportFinished While In Remote Configuration
			ELSIF udiStatus2 = 2936 THEN
				udiStatus2	:= 10125;	//Receive CurrentConfiguration While In Remote Configuration
			ELSIF udiStatus2 = 2937 THEN
				udiStatus2	:= 10126;	//Receive BoardForecast While In Remote Configuration
			ELSIF udiStatus2 = 2938 THEN
				udiStatus2	:= 10127;	//Receive QueryBoardInfo While In Remote Configuration
			ELSIF udiStatus2 = 2939 THEN
				udiStatus2	:= 10128;	//Receive SendBoardInfo While In Remote Configuration
			END_IF

			fHermesAddOneMsgSend(ADR(a_eMsgSend) , ADR(udiMsgSendBffr) , HermesMsgTypeNotification);

			tyNotificationSnd.tyAvl.bSeverity			:= TRUE;
			tyNotificationSnd.tyAvl.bNotificationCode	:= TRUE;
			tyNotificationSnd.tyAvl.bDescription		:= TRUE;
			tyNotificationSnd.tyData.eSeverity			:= HermesSeverityFatalError;
			tyNotificationSnd.tyData.iNotificationCode	:= UDINT_TO_INT(udiStatus2);
			tyNotificationSnd.tyData.sDescription		:= a_tyAlmText[udiStatus2].sAlmText;

		END_IF

	END_IF

END_ACTION
```

#### Act_Background_ChkParamRcv.st - Do Not Change!!!
```iecst
(** 2019-05-04 **)
ACTION Act_Background_ChkParamRcv:

//	IF eStatus2 <> Error THEN

		//Check Parameter Receive
//		IF tyMsgTypeRcv.bSetConfiguration = TRUE THEN

//				fHermesAddOneMsgSend(ADR(a_eMsgSend) , ADR(udiMsgSendBffr) , HermesMsgTypeNotification);
//
//				tyNotificationSnd.tyAvl.bSeverity			:= TRUE;
//				tyNotificationSnd.tyAvl.bNotificationCode	:= TRUE;
//				tyNotificationSnd.tyAvl.bDescription		:= TRUE;
//				tyNotificationSnd.tyData.eSeverity			:= HermesSeverityFatalError;
//				tyNotificationSnd.tyData.iNotificationCode	:= 4;
//				tyNotificationSnd.tyData.sDescription		:= a_tyAlmText[udiStatus2].sAlmText;

//		END_IF
//	END_IF

END_ACTION
```

#### Act_Background_UpdtConfig.st - Do Not Change!!!
```iecst
(** 2021-08-01 **)
ACTION Act_Background_UpdtConfig:

	IF eStatus2 <> Error THEN

		IF tyMsgTypeRcv.bSetConfiguration = TRUE THEN

			tySetConfiguration.tyAvl.bMachineId						:= tySetConfigurationRcv.tyAvl.bMachineId;
			tySetConfiguration.tyAvl.bSupervisorySystemPort			:= tySetConfigurationRcv.tyAvl.bSupervisorySystemPort;
			tySetConfiguration.tyAvl.bUpstreamConfigurations		:= tySetConfigurationRcv.tyAvl.bUpstreamConfigurations;
			tySetConfiguration.tyAvl.bDownstreamConfigurations		:= tySetConfigurationRcv.tyAvl.bDownstreamConfigurations;
			tySetConfiguration.tyAvl.iUpstreamConfigurations		:= tySetConfigurationRcv.tyAvl.iUpstreamConfigurations;
			tySetConfiguration.tyAvl.iDownstreamConfigurations		:= tySetConfigurationRcv.tyAvl.iDownstreamConfigurations;
			tySetConfiguration.tyAvl.a_tyUpstreamConfigurations		:= tySetConfigurationRcv.tyAvl.a_tyUpstreamConfigurations;
			tySetConfiguration.tyAvl.a_tyDownstreamConfigurations	:= tySetConfigurationRcv.tyAvl.a_tyDownstreamConfigurations;

			tySetConfiguration.tyData.sMachineId					:= tySetConfigurationRcv.tyData.sMachineId;
			tySetConfiguration.tyData.uiSupervisorySystemPort		:= tySetConfigurationRcv.tyData.uiSupervisorySystemPort;
			tySetConfiguration.tyData.a_tyUpstreamConfigurations	:= tySetConfigurationRcv.tyData.a_tyUpstreamConfigurations;
			tySetConfiguration.tyData.a_tyDownstreamConfigurations	:= tySetConfigurationRcv.tyData.a_tyDownstreamConfigurations;

			udiTargetAddress := ADR(tySetConfiguration.tyData.a_tyUpstreamConfigurations[0].iUpstreamLaneId); //Start address
			udiSizeAddress   := SIZEOF(tySetConfiguration.tyData.a_tyUpstreamConfigurations[0]); //Size of one array

			udiTargetAddress1 := ADR(tySetConfiguration.tyData.a_tyDownstreamConfigurations[0].iDownstreamLaneId); //Start address
			udiSizeAddress1   := SIZEOF(tySetConfiguration.tyData.a_tyDownstreamConfigurations[0]); //Size of one array

			FOR k := 0 TO c_diHermesConfigMaxIdx DO //Max configuration

				IF memcmp((udiTargetAddress)+(k*udiSizeAddress), ADR(j) , 1) = 0 THEN

					bFoundIndexUS1	:= TRUE;
					udiFoundIndexUS1  := k;

					tySetConfigurationModified.tyData.a_tyUpstreamConfigurations[0].iUpstreamLaneId	        := tySetConfiguration.tyData.a_tyUpstreamConfigurations[udiFoundIndexUS1].iUpstreamLaneId;
					tySetConfigurationModified.tyData.a_tyUpstreamConfigurations[0].sHostAddress	        := tySetConfiguration.tyData.a_tyUpstreamConfigurations[udiFoundIndexUS1].sHostAddress;
					tySetConfigurationModified.tyData.a_tyUpstreamConfigurations[0].sUpstreamInterfaceId	:= tySetConfiguration.tyData.a_tyUpstreamConfigurations[udiFoundIndexUS1].sUpstreamInterfaceId;
					tySetConfigurationModified.tyData.a_tyUpstreamConfigurations[0].uiPort              	:= tySetConfiguration.tyData.a_tyUpstreamConfigurations[udiFoundIndexUS1].uiPort;

				ELSIF memcmp((udiTargetAddress)+(k*udiSizeAddress), ADR(jj) , 1) = 0 THEN

					bFoundIndexUS2	:= TRUE;
					udiFoundIndexUS2  := k;

					tySetConfigurationModified.tyData.a_tyUpstreamConfigurations[1].iUpstreamLaneId	        := tySetConfiguration.tyData.a_tyUpstreamConfigurations[udiFoundIndexUS2].iUpstreamLaneId;
					tySetConfigurationModified.tyData.a_tyUpstreamConfigurations[1].sHostAddress	        := tySetConfiguration.tyData.a_tyUpstreamConfigurations[udiFoundIndexUS2].sHostAddress;
					tySetConfigurationModified.tyData.a_tyUpstreamConfigurations[1].sUpstreamInterfaceId	:= tySetConfiguration.tyData.a_tyUpstreamConfigurations[udiFoundIndexUS2].sUpstreamInterfaceId;
					tySetConfigurationModified.tyData.a_tyUpstreamConfigurations[1].uiPort              	:= tySetConfiguration.tyData.a_tyUpstreamConfigurations[udiFoundIndexUS2].uiPort;

				ELSIF memcmp((udiTargetAddress)+(k*udiSizeAddress), ADR(jjj) , 1) = 0 THEN

					bFoundIndexUS3	:= TRUE;
					udiFoundIndexUS3  := k;

					tySetConfigurationModified.tyData.a_tyUpstreamConfigurations[2].iUpstreamLaneId	        := tySetConfiguration.tyData.a_tyUpstreamConfigurations[udiFoundIndexUS3].iUpstreamLaneId;
					tySetConfigurationModified.tyData.a_tyUpstreamConfigurations[2].sHostAddress	        := tySetConfiguration.tyData.a_tyUpstreamConfigurations[udiFoundIndexUS3].sHostAddress;
					tySetConfigurationModified.tyData.a_tyUpstreamConfigurations[2].sUpstreamInterfaceId	:= tySetConfiguration.tyData.a_tyUpstreamConfigurations[udiFoundIndexUS3].sUpstreamInterfaceId;
					tySetConfigurationModified.tyData.a_tyUpstreamConfigurations[2].uiPort              	:= tySetConfiguration.tyData.a_tyUpstreamConfigurations[udiFoundIndexUS3].uiPort;

				ELSIF memcmp((udiTargetAddress)+(k*udiSizeAddress), ADR(jjjj) , 1) = 0 THEN

					bFoundIndexUS4	:= TRUE;
					udiFoundIndexUS4  := k;

					tySetConfigurationModified.tyData.a_tyUpstreamConfigurations[3].iUpstreamLaneId	        := tySetConfiguration.tyData.a_tyUpstreamConfigurations[udiFoundIndexUS3].iUpstreamLaneId;
					tySetConfigurationModified.tyData.a_tyUpstreamConfigurations[3].sHostAddress	        := tySetConfiguration.tyData.a_tyUpstreamConfigurations[udiFoundIndexUS3].sHostAddress;
					tySetConfigurationModified.tyData.a_tyUpstreamConfigurations[3].sUpstreamInterfaceId	:= tySetConfiguration.tyData.a_tyUpstreamConfigurations[udiFoundIndexUS3].sUpstreamInterfaceId;
					tySetConfigurationModified.tyData.a_tyUpstreamConfigurations[3].uiPort              	:= tySetConfiguration.tyData.a_tyUpstreamConfigurations[udiFoundIndexUS3].uiPort;

				END_IF

			END_FOR

			FOR kk := 0 TO c_diHermesConfigMaxIdx DO //Max configuration

				IF memcmp((udiTargetAddress1)+(kk*udiSizeAddress1), ADR(j) , 1) = 0 THEN

					bFoundIndexDS1	:= TRUE;
					udiFoundIndexDS1  := kk;

					tySetConfigurationModified.tyData.a_tyDownstreamConfigurations[0].iDownstreamLaneId	        := tySetConfiguration.tyData.a_tyDownstreamConfigurations[udiFoundIndexDS1].iDownstreamLaneId;
					tySetConfigurationModified.tyData.a_tyDownstreamConfigurations[0].sClientAddress	        := tySetConfiguration.tyData.a_tyDownstreamConfigurations[udiFoundIndexDS1].sClientAddress;
					tySetConfigurationModified.tyData.a_tyDownstreamConfigurations[0].sDownstreamInterfaceId	:= tySetConfiguration.tyData.a_tyDownstreamConfigurations[udiFoundIndexDS1].sDownstreamInterfaceId;
					tySetConfigurationModified.tyData.a_tyDownstreamConfigurations[0].uiPort                 	:= tySetConfiguration.tyData.a_tyDownstreamConfigurations[udiFoundIndexDS1].uiPort;

				ELSIF memcmp((udiTargetAddress1)+(kk*udiSizeAddress1), ADR(jj) , 1) = 0 THEN

					bFoundIndexDS2	:= TRUE;
					udiFoundIndexDS2  := kk;

					tySetConfigurationModified.tyData.a_tyDownstreamConfigurations[1].iDownstreamLaneId	        := tySetConfiguration.tyData.a_tyDownstreamConfigurations[udiFoundIndexDS2].iDownstreamLaneId;
					tySetConfigurationModified.tyData.a_tyDownstreamConfigurations[1].sClientAddress	        := tySetConfiguration.tyData.a_tyDownstreamConfigurations[udiFoundIndexDS2].sClientAddress;
					tySetConfigurationModified.tyData.a_tyDownstreamConfigurations[1].sDownstreamInterfaceId	:= tySetConfiguration.tyData.a_tyDownstreamConfigurations[udiFoundIndexDS2].sDownstreamInterfaceId;
					tySetConfigurationModified.tyData.a_tyDownstreamConfigurations[1].uiPort                 	:= tySetConfiguration.tyData.a_tyDownstreamConfigurations[udiFoundIndexDS2].uiPort;

				ELSIF memcmp((udiTargetAddress1)+(kk*udiSizeAddress1), ADR(jjj) , 1) = 0 THEN

					bFoundIndexDS3	:= TRUE;
					udiFoundIndexDS3  := kk;

					tySetConfigurationModified.tyData.a_tyDownstreamConfigurations[2].iDownstreamLaneId	        := tySetConfiguration.tyData.a_tyDownstreamConfigurations[udiFoundIndexDS3].iDownstreamLaneId;
					tySetConfigurationModified.tyData.a_tyDownstreamConfigurations[2].sClientAddress	        := tySetConfiguration.tyData.a_tyDownstreamConfigurations[udiFoundIndexDS3].sClientAddress;
					tySetConfigurationModified.tyData.a_tyDownstreamConfigurations[2].sDownstreamInterfaceId	:= tySetConfiguration.tyData.a_tyDownstreamConfigurations[udiFoundIndexDS3].sDownstreamInterfaceId;
					tySetConfigurationModified.tyData.a_tyDownstreamConfigurations[2].uiPort                 	:= tySetConfiguration.tyData.a_tyDownstreamConfigurations[udiFoundIndexDS3].uiPort;

				ELSIF memcmp((udiTargetAddress1)+(kk*udiSizeAddress1), ADR(jjjj) , 1) = 0 THEN

					bFoundIndexDS4	:= TRUE;
					udiFoundIndexDS4  := kk;

					tySetConfigurationModified.tyData.a_tyDownstreamConfigurations[3].iDownstreamLaneId	        := tySetConfiguration.tyData.a_tyDownstreamConfigurations[udiFoundIndexDS4].iDownstreamLaneId;
					tySetConfigurationModified.tyData.a_tyDownstreamConfigurations[3].sClientAddress	        := tySetConfiguration.tyData.a_tyDownstreamConfigurations[udiFoundIndexDS4].sClientAddress;
					tySetConfigurationModified.tyData.a_tyDownstreamConfigurations[3].sDownstreamInterfaceId	:= tySetConfiguration.tyData.a_tyDownstreamConfigurations[udiFoundIndexDS4].sDownstreamInterfaceId;
					tySetConfigurationModified.tyData.a_tyDownstreamConfigurations[3].uiPort                 	:= tySetConfiguration.tyData.a_tyDownstreamConfigurations[udiFoundIndexDS4].uiPort;
				END_IF

			END_FOR

			tySetConfigurationModified.tyAvl.bMachineId				        := tySetConfiguration.tyAvl.bMachineId;
			tySetConfigurationModified.tyAvl.bSupervisorySystemPort			:= tySetConfiguration.tyAvl.bSupervisorySystemPort;
			tySetConfigurationModified.tyAvl.bUpstreamConfigurations		:= tySetConfiguration.tyAvl.bUpstreamConfigurations;
			tySetConfigurationModified.tyAvl.bDownstreamConfigurations		:= tySetConfiguration.tyAvl.bDownstreamConfigurations;
			tySetConfigurationModified.tyAvl.iUpstreamConfigurations		:= tySetConfiguration.tyAvl.iUpstreamConfigurations;
			tySetConfigurationModified.tyAvl.iDownstreamConfigurations		:= tySetConfiguration.tyAvl.iDownstreamConfigurations;
			tySetConfigurationModified.tyAvl.a_tyUpstreamConfigurations		:= tySetConfiguration.tyAvl.a_tyUpstreamConfigurations;
			tySetConfigurationModified.tyAvl.a_tyDownstreamConfigurations	:= tySetConfiguration.tyAvl.a_tyDownstreamConfigurations;

			tySetConfigurationModified.tyData.sMachineId					:= tySetConfiguration.tyData.sMachineId;
			tySetConfigurationModified.tyData.uiSupervisorySystemPort		:= tySetConfiguration.tyData.uiSupervisorySystemPort;

			IF bUpdateUIData = FALSE THEN
				bWriteConfig := TRUE;
				tyMsgTypeRcv.bSetConfiguration	:= FALSE;
			END_IF

		END_IF

	END_IF

END_ACTION
```

#### Act_Background_SendConfig.st - Do Not Change!!!
```iecst
(** 2021-08-01 **)
ACTION Act_Background_SendConfig:

	IF eStatus1 <> Error THEN

		IF tyMsgTypeRcv.bGetConfiguration = TRUE THEN

			IF bWriteConfig = FALSE AND bUpdateUIData = FALSE THEN

				tyCurrentConfigurationSnd.tyData.sMachineId			                        		            := p_sMcId;
				tyCurrentConfigurationSnd.tyData.uiSupervisorySystemPort	                                 	:= p_tyHermesConfiguration.tySvyParam.uiSvySvstemPort;

				FOR i := 0 TO (p_iInput-1) DO
					tyCurrentConfigurationSnd.tyData.a_tyUpstreamConfigurations[i].iUpstreamLaneId	            := p_tyHermesConfiguration.a_tyUSParam[i].iLaneID;
					tyCurrentConfigurationSnd.tyData.a_tyUpstreamConfigurations[i].sHostAddress	                := p_tyHermesConfiguration.a_tyUSParam[i].sHostAddress;
					tyCurrentConfigurationSnd.tyData.a_tyUpstreamConfigurations[i].sUpstreamInterfaceId        	:= p_tyHermesConfiguration.a_tyUSParam[i].sUpstreamInterfaceId;
					tyCurrentConfigurationSnd.tyData.a_tyUpstreamConfigurations[i].uiPort                  	    := p_tyHermesConfiguration.a_tyUSParam[i].uiHostPort;
				END_FOR

				FOR i := 0 TO (p_iOutput-1) DO
					tyCurrentConfigurationSnd.tyData.a_tyDownstreamConfigurations[i].iDownstreamLaneId	        := p_tyHermesConfiguration.a_tyDSParam[i].iLaneID;
					tyCurrentConfigurationSnd.tyData.a_tyDownstreamConfigurations[i].sClientAddress	            := p_tyHermesConfiguration.a_tyDSParam[i].sClientAddress;
					tyCurrentConfigurationSnd.tyData.a_tyDownstreamConfigurations[i].sDownstreamInterfaceId	    := p_tyHermesConfiguration.a_tyDSParam[i].sDownstreamInterfaceId;
					tyCurrentConfigurationSnd.tyData.a_tyDownstreamConfigurations[i].uiPort                 	:= p_tyHermesConfiguration.a_tyDSParam[i].uiSvrPort;
			    END_FOR

				tyCurrentConfigurationSnd.tyAvl.bMachineId					                                	:= tyCurrentConfigurationSnd.tyData.sMachineId <> '';
				tyCurrentConfigurationSnd.tyAvl.bSupervisorySystemPort		                                 	:= tyCurrentConfigurationSnd.tyData.uiSupervisorySystemPort <> 0;
				tyCurrentConfigurationSnd.tyAvl.bUpstreamConfigurations	                                     	:= TRUE;
				tyCurrentConfigurationSnd.tyAvl.bDownstreamConfigurations	                                 	:= TRUE;
				tyCurrentConfigurationSnd.tyAvl.iUpstreamConfigurations	                                     	:= p_iInput;
				tyCurrentConfigurationSnd.tyAvl.iDownstreamConfigurations	   	                                := p_iOutput;

				FOR i := 0 TO (p_iInput-1) DO
					tyCurrentConfigurationSnd.tyAvl.a_tyUpstreamConfigurations[i].bUpstreamLaneId	            := tyCurrentConfigurationSnd.tyData.a_tyUpstreamConfigurations[i].iUpstreamLaneId <>0;
					tyCurrentConfigurationSnd.tyAvl.a_tyUpstreamConfigurations[i].bHostAddress		            := tyCurrentConfigurationSnd.tyData.a_tyUpstreamConfigurations[i].sHostAddress <>'';
					tyCurrentConfigurationSnd.tyAvl.a_tyUpstreamConfigurations[i].bUpstreamInterfaceId	        := tyCurrentConfigurationSnd.tyData.a_tyUpstreamConfigurations[i].sUpstreamInterfaceId <>'';
					tyCurrentConfigurationSnd.tyAvl.a_tyUpstreamConfigurations[i].bPort		                    := tyCurrentConfigurationSnd.tyData.a_tyUpstreamConfigurations[i].uiPort <>0;
				END_FOR

				FOR i := 0 TO (p_iOutput-1) DO
					tyCurrentConfigurationSnd.tyAvl.a_tyDownstreamConfigurations[i].bDownstreamLaneId	    	:= tyCurrentConfigurationSnd.tyData.a_tyDownstreamConfigurations[i].iDownstreamLaneId <>0;
					tyCurrentConfigurationSnd.tyAvl.a_tyDownstreamConfigurations[i].bClientAddress		        := tyCurrentConfigurationSnd.tyData.a_tyDownstreamConfigurations[i].sClientAddress <>'';
					tyCurrentConfigurationSnd.tyAvl.a_tyDownstreamConfigurations[i].bDownstreamInterfaceId	    := tyCurrentConfigurationSnd.tyData.a_tyDownstreamConfigurations[i].sDownstreamInterfaceId <>'';
					tyCurrentConfigurationSnd.tyAvl.a_tyDownstreamConfigurations[i].bPort		                := tyCurrentConfigurationSnd.tyData.a_tyDownstreamConfigurations[i].uiPort <>0;
				END_FOR

				fHermesAddOneMsgSend(ADR(a_eMsgSend) , ADR(udiMsgSendBffr) , HermesMsgTypeCurrConfiguration);

				tyMsgTypeRcv.bGetConfiguration	:= FALSE;

			END_IF

		END_IF

	END_IF

END_ACTION
```

#### Act_Background_NotificationSnd.st - Do Not Change!!!
```iecst
(** 2021-08-01 **)
ACTION Act_Background_NotificationSnd:

	IF a_eMsgSend[0] = HermesMsgTypeNotification THEN
		bRstConnection	:= fHermesNotificationRstConn(tyNotificationSnd) OR bRstConnection;
	END_IF

END_ACTION
```

#### Act_Background_TCPSend.st - Do Not Change!!!
```iecst
(** 2021-08-01 **)
ACTION Act_Background_TCPSend:

	//Message Send (Generate XML Message)
	IF a_eMsgSend[0] <> HermesMsgTypeNA THEN

		IF a_eMsgSend[0] = HermesMsgTypeCheckAlive THEN
			eStatus1	:= Error;
			udiStatus1	:= 10106;	//Check Alive Request To Send From Remote Hermes

		ELSIF a_eMsgSend[0] = HermesMsgTypeCheckAlivePing THEN
			eStatus1	:= Error;
			udiStatus1	:= 10107;	//Check Alive Ping Request To Send From Remote Hermes

		ELSIF a_eMsgSend[0] = HermesMsgTypeCheckAlivePong THEN
			eStatus1	:= Error;
			udiStatus1	:= 10108;	//Check Alive Pong Request To Send From Remote Hermes

		ELSIF a_eMsgSend[0] = HermesMsgTypeServiceDescription THEN
			eStatus1	:= Error;
			udiStatus1	:= 10130;	//Service Description Request To Send From Remote Hermes

		ELSIF a_eMsgSend[0] = HermesMsgTypeNotification THEN
			fHermesFormNotification(ADR(a_tyXMLTableDataSnd) , p_tyDTStructure , tyNotificationSnd);
			fTableConvertToXML(ADR(sSnd) , ADR(udiSndMsgLen) , SIZEOF(sSnd) , ADR(a_tyXMLTableDataSnd) , ADR(a_tyXMLTableDataSnd[0].sTitle) , ADR(a_tyXMLTableDataSnd[0].sValue) , ADR(a_tyXMLTableDataSnd[0].uiSize) , SIZEOF(a_tyXMLTableDataSnd[0]) , 14);

		ELSIF a_eMsgSend[0] = HermesMsgTypeBoardAvailable THEN
			eStatus1	:= Error;
			udiStatus1	:= 10131;	//Board Available Request To Send From Remote Hermes

		ELSIF a_eMsgSend[0] = HermesMsgTypeRevokeBoardAvl THEN
			eStatus1	:= Error;
			udiStatus1	:= 10132;	//Revoke Board Available Request To Send From Remote Hermes

		ELSIF a_eMsgSend[0] = HermesMsgTypeMachineReady THEN
			eStatus1	:= Error;
			udiStatus1	:= 10135;	//Machine Ready Request To Send From Remote Hermes

		ELSIF a_eMsgSend[0] = HermesMsgTypeRevokeMachineReady THEN
			eStatus1	:= Error;
			udiStatus1	:= 10136;	//Revoke Machine Ready Request To Send From Remote Hermes

		ELSIF a_eMsgSend[0] = HermesMsgTypeStartTransport THEN
			eStatus1	:= Error;
			udiStatus1	:= 10137;	//Start Transport Request To Send From Remote Hermes

		ELSIF a_eMsgSend[0] = HermesMsgTypeStopTransport THEN
			eStatus1	:= Error;
			udiStatus1	:= 10133;	//Stop Transport Request To Send From Remote Hermes

		ELSIF a_eMsgSend[0] = HermesMsgTypeTransportFinished THEN
			eStatus1	:= Error;
			udiStatus1	:= 10134;	//Transport Finished Request To Send From Remote Hermes

		ELSIF a_eMsgSend[0] = HermesMsgTypeSetConfiguration THEN
			eStatus1	:= Error;
			udiStatus1	:= 10138;	//Set Configuration Request To Send From Remote Hermes

		ELSIF a_eMsgSend[0] = HermesMsgTypeGetConfiguration THEN
			eStatus1	:= Error;
			udiStatus1	:= 10139;	//Get Configuration Request To Send From Remote Hermes

		ELSIF a_eMsgSend[0] = HermesMsgTypeCurrConfiguration THEN
			fHermesFormCurrentConfiguration(ADR(a_tyXMLTableDataSnd) , p_tyDTStructure , tyCurrentConfigurationSnd);
			fTableConvertToXML(ADR(sSnd) , ADR(udiSndMsgLen) , SIZEOF(sSnd) , ADR(a_tyXMLTableDataSnd) , ADR(a_tyXMLTableDataSnd[0].sTitle) , ADR(a_tyXMLTableDataSnd[0].sValue) , ADR(a_tyXMLTableDataSnd[0].uiSize) , SIZEOF(a_tyXMLTableDataSnd[0]) , 200);
			//10140

		ELSIF a_eMsgSend[0] = HermesMsgTypeBoardForecast THEN
			eStatus1	:= Error;
			udiStatus1	:= 10141;	//Board Forecast Request To Send From Remote Hermes

		ELSIF a_eMsgSend[0] = HermesMsgTypeQueryBoardInfo THEN
			eStatus1	:= Error;
			udiStatus1	:= 10142;	//Query Board Info Request To Send From Remote Hermes

		ELSIF a_eMsgSend[0] = HermesMsgTypeSendBoardInfo THEN
			eStatus1	:= Error;
			udiStatus1	:= 10159;	//Send Board Info Request To Send From Remote Hermes

		ELSIF a_eMsgSend[0] = HermesMsgTypeQueryWorkOrderInfo THEN
			eStatus1	:= Error;
			udiStatus1	:= 10160;	//Query Work Order Info Request To Send From Remote Hermes

		ELSIF a_eMsgSend[0] = HermesMsgTypeSendWorkOrderInfo THEN
			eStatus1	:= Error;
			udiStatus1	:= 10161;	//Send Work Order Info Request To Send From Remote Hermes

		ELSIF a_eMsgSend[0] = HermesMsgTypeBoardArrived THEN
			eStatus1	:= Error;
			udiStatus1	:= 10162;	//BoardArrived Request To Send From Remote Hermes

		ELSIF a_eMsgSend[0] = HermesMsgTypeBoardDeparted THEN
			eStatus1	:= Error;
			udiStatus1	:= 10163;	//BoardDeparted Request To Send From Remote Hermes

		END_IF

		//Message Send
		fbSend.udiTCPIdent	:= udiClntIdent;
		fbSend.udiSndSize	:= udiSndMsgLen;
		fbSend(bEn := TRUE);

		IF fbSend.udiStatus = 0 THEN

			fLogDTConvert(ADR(sDT) , p_dtCurrDT);
			memset(ADR(a_sLogList[udiLogCntr]) , 0 , SIZEOF(a_sLogList[udiLogCntr]));
			memcpy(ADR(a_sLogList[udiLogCntr]) + LEN(a_sLogList[udiLogCntr]) , ADR(sDT) , LEN(sDT));
			memcpy(ADR(a_sLogList[udiLogCntr]) + LEN(a_sLogList[udiLogCntr]) , ADR('$r$n') , LEN('$r$n'));
			memcpy(ADR(a_sLogList[udiLogCntr]) + LEN(a_sLogList[udiLogCntr]) , ADR('SND_TO_RMT$r$n') , LEN('SND_TO_RMT$r$n'));
			memcpy(ADR(a_sLogList[udiLogCntr]) + LEN(a_sLogList[udiLogCntr]) , ADR(sSnd) , LEN(sSnd));
			memcpy(ADR(a_sLogList[udiLogCntr]) + LEN(a_sLogList[udiLogCntr]) , ADR('$r$n$r$n') , LEN('$r$n$r$n'));

			udiLogCntr	:= udiLogCntr + 1;
			IF udiLogCntr = 11 THEN
				udiLogCntr	:= 1;
			END_IF

			Act_Background_NotificationSnd;
			fHermesRmvOneMsgSend(ADR(a_eMsgSend) , ADR(udiMsgSendBffr));

			fbSend(bEn := FALSE);

		ELSIF fbSend.udiStatus = 2321 THEN
			bRstConnection	:= TRUE;

		ELSIF fbSend.udiStatus < 65534 THEN
			eStatus1	:= Error;

			IF fbSend.udiStatus = 2300 THEN
				udiStatus1	:= 10143;	//Invalid Ident While Sending Data
			ELSIF fbSend.udiStatus = 2320 THEN
				udiStatus1	:= 10144;	//TCP Retry Send Data Error While Sending Data
			ELSIF fbSend.udiStatus = 2322 THEN
				udiStatus1	:= 10145;	//TCP Send Data Error
			ELSE
				udiStatus1	:= fbSend.udiStatus;
			END_IF

		END_IF

	END_IF

END_ACTION
```

#### Act_Background_TCPCloseSvr.st - Do Not Change!!!
```iecst
(** 2021-08-01 **)
ACTION Act_Background_TCPCloseSvr:

	//Close Server Connection
	fbCloseSvr.udiTCPIdent	:= udiSvrIdent;
	fbCloseSvr(bEn := TRUE);

	IF fbCloseSvr.udiStatus = 0 THEN
		udiSvrIdent		:= 0;
		fbCloseSvr(bEn := FALSE);

	ELSIF fbCloseSvr.udiStatus < 65534 THEN
		udiSvrIdent		:= 0;
		eStatus1		:= Error;

		IF fbCloseSvr.udiStatus = 2300 THEN
			udiStatus1	:= 10146;	//Invalid Ident While Closing TCP
		ELSIF fbCloseSvr.udiStatus = 2310 THEN
			udiStatus1	:= 10147;	//Closing TCP Error
		ELSE
			udiStatus1	:= fbCloseSvr.udiStatus;
		END_IF

	END_IF

END_ACTION
```

#### Act_Background_TCPCloseClnt.st - Do Not Change!!!
```iecst
(** 2021-08-01 **)
ACTION Act_Background_TCPCloseClnt:

	//Close Server Connection
	fbCloseClnt.udiTCPIdent	:= udiClntIdent;
	fbCloseClnt(bEn := TRUE);

	IF fbCloseClnt.udiStatus = 0 THEN
		udiClntIdent	:= 0;
		fbCloseClnt(bEn := FALSE);

	ELSIF fbCloseClnt.udiStatus < 65534 THEN
		udiClntIdent	:= 0;
		eStatus1		:= Error;

		IF fbCloseClnt.udiStatus = 2300 THEN
			udiStatus1	:= 10154;	//Invalid Ident While Closing TCP
		ELSIF fbCloseClnt.udiStatus = 2310 THEN
			udiStatus1	:= 10155;	//Closing TCP Error
		ELSE
			udiStatus1	:= fbCloseClnt.udiStatus;
		END_IF

	END_IF

END_ACTION
```

#### Act_Background_Stop.st - Do Not Change!!!
```iecst
(** 2021-08-01 **)
ACTION Act_Background_Stop:

	IF bStop = TRUE THEN //Note: Rmt Station only connect to our Server(udiClntIdent >0) when sending msg to us, after that udiClntIdent will bcome 0. So notification cannot be send out.

		bRstConnection	:= TRUE;

		IF udiSvrIdent = 0 THEN

			bRun	:= FALSE;

		END_IF

	END_IF

END_ACTION
```

#### Act_Background_Err.st - Do Not Change!!!
```iecst
(** 2021-08-01 **)
ACTION Act_Background_Err:

END_ACTION
```

#### Act_Main_Disable.st - Do Not Change!!!
```iecst
(** 2021-08-01 **)
ACTION Act_Main_Disable:

	bConnected		:= FALSE;

END_ACTION
```

#### Act_Alarm.st - Do Not Change!!!
```iecst
(** 2021-08-01 **)
ACTION Act_Alarm: //General

	//Error
	IF EDGEPOS(eStatus = Error) THEN

		tyAlmData.sProgNm		:= p_sProgNm;
		tyAlmData.udiCode		:= udiStatus;
		tyAlmData.eSeverity		:= AlmSeverityError;
		tyAlmData.udiRunTime	:= tyAlmData.udiRunTime + 1;
		tyAlmData.bAlm			:= TRUE;
		tyAlmData.udiModuleNum  := udiModuleNum;
		g_sRmtHermesProgNm		:= p_sProgNm;

		//Get Error Message
		IF tyAlmData.udiCode < 10000 OR tyAlmData.udiCode > 10199 THEN
			tyAlmData.sAlmMsg	:= 'Unknown';
			tyAlmData.sRcyMsg	:= 'Unknown';
		ELSE
			tyAlmData.sAlmMsg	:= a_tyAlmText[tyAlmData.udiCode].sAlmText;
			tyAlmData.sRcyMsg	:= a_tyAlmText[tyAlmData.udiCode].sRcyText;
		END_IF

		sStatTxt	:= tyAlmData.sAlmMsg;

	ELSIF bRstErr AND (tyAlmData.udiCode <> 0) THEN

		tyAlmData.udiCode	:= 0;
		tyAlmData.eSeverity	:= AlmSeverityNA;
		tyAlmData.sAlmMsg	:= '';
		tyAlmData.sRcyMsg	:= '';
		tyAlmData.bAlm			:= FALSE;
		sStatTxt	:= a_sStatText[eStat];

	END_IF

END_ACTION
```

#### Act_Alarm1.st - Do Not Change!!!
```iecst
(** 2021-08-01 **)
ACTION Act_Alarm1:

	//Error
	IF EDGEPOS(eStatus1 = Error) THEN

		tyAlmData1.sProgNm		:= p_sProgNm;
		tyAlmData1.udiCode		:= udiStatus1;
		tyAlmData1.eSeverity	:= AlmSeverityError;
		tyAlmData1.udiRunTime	:= tyAlmData1.udiRunTime + 1;
		tyAlmData1.bAlm			:= TRUE;
		tyAlmData1.udiModuleNum  := udiModuleNum;
		g_sRmtHermesProgNm		:= p_sProgNm;
		//Get Error Message
		IF tyAlmData1.udiCode < 10000 OR tyAlmData1.udiCode > 10199 THEN
			tyAlmData1.sAlmMsg	:= 'Unknown';
			tyAlmData1.sRcyMsg	:= 'Unknown';
		ELSE
			tyAlmData1.sAlmMsg	:= a_tyAlmText[tyAlmData1.udiCode].sAlmText;
			tyAlmData1.sRcyMsg	:= a_tyAlmText[tyAlmData1.udiCode].sRcyText;
		END_IF

		sStatTxt	:= tyAlmData1.sAlmMsg;

	ELSIF bRstErr AND (tyAlmData1.udiCode <> 0) THEN

		tyAlmData1.udiCode		:= 0;
		tyAlmData1.eSeverity	:= AlmSeverityNA;
		tyAlmData1.sAlmMsg		:= '';
		tyAlmData1.sRcyMsg		:= '';
		tyAlmData1.bAlm			:= FALSE;
		sStatTxt	:= a_sStatText[eStat];

	END_IF

END_ACTION
```

#### Act_Alarm2.st - Do Not Change!!!
```iecst
(** 2021-08-01 **)
ACTION Act_Alarm2:

	//Error
	IF EDGEPOS(eStatus2 = Error) THEN

		tyAlmData2.sProgNm		:= p_sProgNm;
		tyAlmData2.udiCode		:= udiStatus2;
		tyAlmData2.eSeverity	:= AlmSeverityError;
		tyAlmData2.udiRunTime	:= tyAlmData2.udiRunTime + 1;
		tyAlmData2.bAlm			:= TRUE;
		tyAlmData2.udiModuleNum  := udiModuleNum;
		g_sRmtHermesProgNm		:= p_sProgNm;
		//Get Error Message
		IF tyAlmData2.udiCode < 10000 OR tyAlmData2.udiCode > 10199 THEN
			tyAlmData2.sAlmMsg	:= 'Unknown';
			tyAlmData2.sRcyMsg	:= 'Unknown';
		ELSE
			tyAlmData2.sAlmMsg	:= a_tyAlmText[tyAlmData2.udiCode].sAlmText;
			tyAlmData2.sRcyMsg	:= a_tyAlmText[tyAlmData2.udiCode].sRcyText;
		END_IF

		sStatTxt	:= tyAlmData2.sAlmMsg;

	ELSIF bRstErr AND (tyAlmData2.udiCode <> 0) THEN

		tyAlmData2.udiCode		:= 0;
		tyAlmData2.eSeverity	:= AlmSeverityNA;
		tyAlmData2.sAlmMsg		:= '';
		tyAlmData2.sRcyMsg		:= '';
		tyAlmData2.bAlm			:= FALSE;
		sStatTxt	:= a_sStatText[eStat];

	END_IF

END_ACTION
```

#### Act_Alarm3.st - Do Not Change!!!
```iecst
(** 2021-08-01 **)
ACTION Act_Alarm3: //fbFileAppend1 Error

	//Error
	IF EDGEPOS(eStatus3 = Error) THEN

		tyAlmData3.sProgNm		:= p_sProgNm;
		tyAlmData3.udiCode		:= udiStatus3;
		tyAlmData3.eSeverity	:= AlmSeverityError;
		tyAlmData3.udiRunTime	:= tyAlmData3.udiRunTime + 1;
		tyAlmData3.bAlm			:= TRUE;
		tyAlmData3.udiModuleNum  := udiModuleNum;
		g_sRmtHermesProgNm		:= p_sProgNm;
		//Get Error Message
		IF tyAlmData3.udiCode < 10000 OR tyAlmData3.udiCode > 10199 THEN
			tyAlmData3.sAlmMsg	:= 'Unknown';
			tyAlmData3.sRcyMsg	:= 'Unknown';
		ELSE
			tyAlmData3.sAlmMsg	:= a_tyAlmText[tyAlmData3.udiCode].sAlmText;
			tyAlmData3.sRcyMsg	:= a_tyAlmText[tyAlmData3.udiCode].sRcyText;
		END_IF

		sStatTxt	:= tyAlmData3.sAlmMsg;

	ELSIF bRstErr AND (tyAlmData3.udiCode <> 0) THEN

		tyAlmData3.udiCode		:= 0;
		tyAlmData3.eSeverity	:= AlmSeverityNA;
		tyAlmData3.sAlmMsg		:= '';
		tyAlmData3.sRcyMsg		:= '';
		tyAlmData3.bAlm			:= FALSE;
		sStatTxt	:= a_sStatText[eStat];

	END_IF

END_ACTION
```

#### InputRef.var - Do Not Change!!!
```iecst
(*2021-08-01*)
(**)
(*General*)
VAR
	p_eAct : REFERENCE TO eHermesAction;
	p_udiRstErr : REFERENCE TO UDINT;
	p_bPrep : REFERENCE TO BOOL;
	p_bEn : REFERENCE TO BOOL;
	p_bDis : REFERENCE TO BOOL;
END_VAR
(**)
(*Configuration*)
VAR
	p_tyParam : REFERENCE TO tyHermesRmtParam;
	p_sIPAddr : REFERENCE TO STRING[15];
	p_tyDTStructure : REFERENCE TO DTStructure;
	p_dtCurrDT : REFERENCE TO DATE_AND_TIME;
	p_sMcId : REFERENCE TO STRING[80];
END_VAR
(**)
(*Input*)
VAR
	p_bRmtPrep : REFERENCE TO BOOL;
	p_bRmtEn : REFERENCE TO BOOL;
	p_udiSndBffrSize : REFERENCE TO UDINT;
	p_udiRcvBffrSize : REFERENCE TO UDINT;
	p_udiAliveIdleTimeInSec : REFERENCE TO UDINT;
	p_udiFileKeepDay : REFERENCE TO UDINT;
	p_sConfigFileName : REFERENCE TO STRING[80];
	p_sProgNm : REFERENCE TO STRING[15];
	p_bNtSettingsLoadDone : REFERENCE TO BOOL;
	p_iInput : REFERENCE TO INT;
	p_iOutput : REFERENCE TO INT;
	p_sInfoMsg : REFERENCE TO STRING[200];
	p_tyHermesConfiguration : REFERENCE TO tyHermesConfiguration;
	p_eHermesStat : REFERENCE TO eHermesAction;
	p_eHermesStatus : REFERENCE TO eFBStatus;
	p_eMcParamStat : REFERENCE TO eMcParamAction;
	p_eMcParamStatus : REFERENCE TO eFBStatus;
END_VAR
```

#### Local.var - Do Not Change!!!
```iecst
(*2021-08-01*)
(**)
(*Local Action, State & Status*)
VAR
	eAct : eHermesAction := HermesActIdle;
	eStat : eHermesAction := HermesActIdle;
	eHermesAct : eHermesAction;
	eMcParamAct : eMcParamAction;
	eMainStatus : eFBStatus := Idle;
	eStatus : eFBStatus := Idle;
	eStatus1 : eFBStatus := Idle;
	eStatus2 : eFBStatus := Idle;
	eStatus3 : eFBStatus := Idle;
	udiStatus : UDINT := 0;
	udiStatus1 : UDINT := 0;
	udiStatus2 : UDINT := 0;
	udiStatus3 : UDINT := 0;
	sStatTxt : STRING[200] := '';
	a_sStatText : ARRAY[0..50] OF STRING[200] := ['Idling','Background Starting Operations','Background Stopping Operations','Deleting Old Log File','Creating Directory','Writing Retain File','Reading Retain File','Saving Configuration',43('')];
END_VAR
(**)
(*Local Alarm*)
VAR
	tyAlmData : tyAlmDat;
	tyAlmData1 : tyAlmDat;
	tyAlmData2 : tyAlmDat;
	tyAlmData3 : tyAlmDat;
	tyInfoData : tyAlmDat;
	sInfoMsg : STRING[200];
	a_tyAlmText : ARRAY[10000..10199] OF tyAlmTxt := [(sAlmText:='Invalid Ident While Creating Server',sRcyText:='Problem Occurred In The TCP/IP Connection. Check The Connection And Try To Reconnect.'),(sAlmText:='Setting Keep Alive Interval Time Error While Creating Server',sRcyText:='Unable To Establish Connection Between Machine. Check For Setting And Resume Operation.'),(sAlmText:='Setting Keep Alive Idle Time Error While Creating Server',sRcyText:='Unable To Establish Connection Between Machine. Check For Setting And Resume Operation.'),(sAlmText:='Setting Keep Alive Count Error While Creating Server',sRcyText:='Unable To Establish Connection Between Machine. Check For Setting And Resume Operation.'),(sAlmText:='Setting Keep Alive Error While Creating Server',sRcyText:='Unable To Establish Connection Between Machine. Check For Setting And Resume Operation.'),(sAlmText:='Setting Receive Buffer Error While Creating Server',sRcyText:='Unable To Establish Connection Between Machine. Check For Setting And Resume Operation.'),(sAlmText:='Setting Send Buffer Error While Creating Server',sRcyText:='Unable To Establish Connection Between Machine. Check For Setting And Resume Operation.'),(sAlmText:='Setting No Waiting Error While Creating Server',sRcyText:='Unable To Establish Connection Between Machine. Check For Setting And Resume Operation.'),(sAlmText:='TCP Open Port Error While Creating Server',sRcyText:='Problem Occurred In The TCP/IP Connection. Check The Connection And Try To Reconnect.'),(sAlmText:='Closing TCP Error While Creating Server',sRcyText:='Problem Occurred In The TCP/IP Connection. Check The Connection And Try To Reconnect.'),(sAlmText:='Invalid Ident While Listening Client',sRcyText:='There Was A Problem Connecting To The Server. The Server May Not Exist or It is Unavailable At This Time. Check The Connection and Try Again.'),(0),(sAlmText:='Listen To Client Error While Listening Client',sRcyText:='There Was A Problem Connecting To The Server. The Server May Not Exist or It is Unavailable At This Time. Check The Connection and Try Again.'),(0),(sAlmText:='Invalid Ident While Receiving Data',sRcyText:='Problem Occurred In The TCP/IP Connection. Check The Connection And Try To Reconnect.'),(sAlmText:='TCP Receive Data Error While Receiving Data',sRcyText:='Problem Occurred In The TCP/IP Connection. Check The Connection And Try To Reconnect.'),(sAlmText:='Receive BoardAvailable While Downstream In Not Connected State',sRcyText:='Receive Illegal Message.'),(sAlmText:='Receive RevokeBoardAvailable While Downstream In Not Connected State',sRcyText:='Receive Illegal Message.'),(sAlmText:='Receive MachineReady While Downstream In Not Connected State',sRcyText:='Receive Illegal Message.'),(sAlmText:='Receive RevokeMachineReady While Downstream In Not Connected State',sRcyText:='Receive Illegal Message.'),(sAlmText:='Receive StartTransport While Downstream In Not Connected State',sRcyText:='Receive Illegal Message.'),(sAlmText:='Receive StopTransport While Downstream In Not Connected State',sRcyText:='Receive Illegal Message.'),(sAlmText:='Receive TransportFinished While Downstream In Not Connected State',sRcyText:='Receive Illegal Message.'),(sAlmText:='Receive BoardForecast While Downstream In Not Connected State',sRcyText:='Receive Illegal Message.'),(sAlmText:='Receive ServiceDescription While Downstream In Service Description State',sRcyText:='Receive Illegal Message.'),(sAlmText:='Receive BoardAvailable While Downstream In Service Description State',sRcyText:='Receive Illegal Message.'),(sAlmText:='Receive RevokeBoardAvailable While Downstream In Service Description State',sRcyText:='Receive Illegal Message.'),(sAlmText:='Receive MachineReady While Downstream In Service Description State',sRcyText:='Receive Illegal Message.'),(sAlmText:='Receive RevokeMachineReady While Downstream In Service Description State',sRcyText:='Receive Illegal Message.'),(sAlmText:='Receive StartTransport While Downstream In Service Description State',sRcyText:='Receive Illegal Message.'),(sAlmText:='Receive StopTransport While Downstream In Service Description State',sRcyText:='Receive Illegal Message.'),(sAlmText:='Receive TransportFinished While Downstream In Service Description State',sRcyText:='Receive Illegal Message.'),(sAlmText:='Receive BoardForecast While Downstream In Service Description State',sRcyText:='Receive Illegal Message.'),(sAlmText:='Receive ServiceDescription While Downstream In Not Available Not Ready State',sRcyText:='Receive Illegal Message.'),(sAlmText:='Receive BoardAvailable While Downstream In Not Available Not Ready State',sRcyText:='Receive Illegal Message.'),(sAlmText:='Receive RevokeBoardAvailable While Downstream In Not Available Not Ready State',sRcyText:='Receive Illegal Message.'),(sAlmText:='Receive RevokeMachineReady While Downstream In Not Available Not Ready State',sRcyText:='Receive Illegal Message.'),(sAlmText:='Receive StartTransport While Downstream In Not Available Not Ready State',sRcyText:='Receive Illegal Message.'),(sAlmText:='Receive StopTransport While Downstream In Not Available Not Ready State',sRcyText:='Receive Illegal Message.'),(sAlmText:='Receive TransportFinished While Downstream In Not Available Not Ready State',sRcyText:='Receive Illegal Message.'),(sAlmText:='Receive BoardForecast While Downstream In Not Available Not Ready State',sRcyText:='Receive Illegal Message.'),(sAlmText:='Receive ServiceDescription While Downstream In Board Available State',sRcyText:='Receive Illegal Message.'),(sAlmText:='Receive BoardAvailable While Downstream In Board Available State',sRcyText:='Receive Illegal Message.'),(sAlmText:='Receive RevokeBoardAvailable While Downstream In Board Available State',sRcyText:='Receive Illegal Message.'),(sAlmText:='Receive RevokeMachineReady While Downstream In Board Available State',sRcyText:='Receive Illegal Message.'),(sAlmText:='Receive StartTransport While Downstream In Board Available State',sRcyText:='Receive Illegal Message.'),(sAlmText:='Receive StopTransport While Downstream In Board Available State',sRcyText:='Receive Illegal Message.'),(sAlmText:='Receive TransportFinished While Downstream In Board Available State',sRcyText:='Receive Illegal Message.'),(sAlmText:='Receive BoardForecast While Downstream In Board Available State',sRcyText:='Receive Illegal Message.'),(sAlmText:='Receive ServiceDescription While Downstream In Machine Ready State',sRcyText:='Receive Illegal Message.'),(sAlmText:='Receive BoardAvailable While Downstream In Machine Ready State',sRcyText:='Receive Illegal Message.'),(sAlmText:='Receive RevokeBoardAvailable While Downstream In Machine Ready State',sRcyText:='Receive Illegal Message.'),(sAlmText:='Receive MachineReady While Downstream In Machine Ready State',sRcyText:='Receive Illegal Message.'),(sAlmText:='Receive StopTransport While Downstream In Machine Ready State',sRcyText:='Receive Illegal Message.'),(sAlmText:='Receive TransportFinished While Downstream In Machine Ready State',sRcyText:='Receive Illegal Message.'),(sAlmText:='Receive BoardForecast While Downstream In Machine Ready State',sRcyText:='Receive Illegal Message.'),(sAlmText:='Receive ServiceDescription While Downstream In Available And Ready State',sRcyText:='Receive Illegal Message.'),(sAlmText:='Receive BoardAvailable While Downstream In Available And Ready State',sRcyText:='Receive Illegal Message.'),(sAlmText:='Receive RevokeBoardAvailable While Downstream In Available And Ready State',sRcyText:='Receive Illegal Message.'),(sAlmText:='Receive MachineReady While Downstream In Available And Ready State',sRcyText:='Receive Illegal Message.'),(sAlmText:='Receive StopTransport While Downstream In Available And Ready State',sRcyText:='Receive Illegal Message.'),(sAlmText:='Receive TransportFinished While Downstream In Available And Ready State',sRcyText:='Receive Illegal Message.'),(sAlmText:='Receive BoardForecast While Downstream In Available And Ready State',sRcyText:='Receive Illegal Message.'),(sAlmText:='Receive ServiceDescription While Downstream In Transporting State',sRcyText:='Receive Illegal Message.'),(sAlmText:='Receive BoardAvailable While Downstream In Transporting State',sRcyText:='Receive Illegal Message.'),(sAlmText:='Receive RevokeBoardAvailable While Downstream In Transporting State',sRcyText:='Receive Illegal Message.'),(sAlmText:='Receive MachineReady While Downstream In Transporting State',sRcyText:='Receive Illegal Message.'),(sAlmText:='Receive RevokeMachineReady While Downstream In Transporting State',sRcyText:='Receive Illegal Message.'),(sAlmText:='Receive StartTransport While Downstream In Transporting State',sRcyText:='Receive Illegal Message.'),(sAlmText:='Receive TransportFinished While Downstream In Transporting State',sRcyText:='Receive Illegal Message.'),(sAlmText:='Receive BoardForecast While Downstream In Transporting State',sRcyText:='Receive Illegal Message.'),(sAlmText:='Receive ServiceDescription While In Transport Finished State',sRcyText:='Receive Illegal Message.'),(sAlmText:='Receive BoardAvailable While In Transport Finished State',sRcyText:='Receive Illegal Message.'),(sAlmText:='Receive RevokeBoardAvailable While In Transport Finished State',sRcyText:='Receive Illegal Message.'),(sAlmText:='Receive MachineReady While In Transport Finished State',sRcyText:='Receive Illegal Message.'),(sAlmText:='Receive RevokeMachineReady While In Transport Finished State',sRcyText:='Receive Illegal Message.'),(sAlmText:='Receive StartTransport While In Transport Finished State',sRcyText:='Receive Illegal Message.'),(sAlmText:='Receive TransportFinished While In Transport Finished State',sRcyText:='Receive Illegal Message.'),(sAlmText:='Receive BoardForecast While In Transport Finished State',sRcyText:='Receive Illegal Message.'),(sAlmText:='Receive ServiceDescription While Downstream In Transport Stopped State',sRcyText:='Receive Illegal Message.'),(sAlmText:='Receive BoardAvailable While Downstream In Transport Stopped State',sRcyText:='Receive Illegal Message.'),(sAlmText:='Receive RevokeBoardAvailable While Downstream In Transport Stopped State',sRcyText:='Receive Illegal Message.'),(sAlmText:='Receive MachineReady While Downstream In Transport Stopped State',sRcyText:='Receive Illegal Message.'),(sAlmText:='Receive RevokeMachineReady While Downstream In Transport Stopped State',sRcyText:='Receive Illegal Message.'),(sAlmText:='Receive StartTransport While Downstream In Transport Stopped State',sRcyText:='Receive Illegal Message.'),(sAlmText:='Receive StopTransport While Downstream In Transport Stopped State',sRcyText:='Receive Illegal Message.'),(sAlmText:='File Open Error While Writing Config File',sRcyText:='An Error Was Encountered While Trying To Open File. Please Contact Nutek For A Possible Solution.'),(sAlmText:='File Create Error While Writing Config File',sRcyText:='An Error Was Encountered While Trying To Create File. Please Contact Nutek For A Possible Solution.'),(sAlmText:='File Write Error While Writing Config File',sRcyText:='An Error Was Encountered While Trying To Write File. Please Contact Nutek For A Possible Solution.'),(sAlmText:='File Close Error While Writing Config File',sRcyText:='An Error Was Encountered While Trying To Close File. Please Contact Nutek For A Possible Solution.'),(sAlmText:='Directory Does Not Exist While Writing Config File',sRcyText:='The Directory Does Not Exist. Please Contact Nutek For A Possible Solution.'),(sAlmText:='File Open Error While Reading Config File',sRcyText:='An Error Was Encountered While Trying To Open File. Please Contact Nutek For A Possible Solution.'),(sAlmText:='File Read Error While Reading Config File',sRcyText:='An Error Was Encountered While Trying To Read File. Please Contact Nutek For A Possible Solution.'),(sAlmText:='File Close Error While Reading Config File',sRcyText:='An Error Was Encountered While Trying To Close File. Please Contact Nutek For A Possible Solution.'),12((0)),(sAlmText:='Check Alive Request To Send From Remote Hermes',sRcyText:='Sending Illegal Message.'),(sAlmText:='Check Alive Ping Request To Send From Remote Hermes',sRcyText:='Sending Illegal Message.'),(sAlmText:='Check Alive Pong Request To Send From Remote Hermes',sRcyText:='Sending Illegal Message.'),(sAlmText:='Receive BoardForecast While Downstream In Transport Stopped State',sRcyText:='Receive Illegal Message.'),(0),(sAlmText:='Get Directory Info Error While Deleting Old Log',sRcyText:='An Error Was Encountered While Getting Directory Info. Please Contact Nutek For A Possible Solution.'),(sAlmText:='Directory Read Error While Deleting Old Log',sRcyText:='An Error Was Encountered While Reading Directory. Please Contact Nutek For A Possible Solution.'),(sAlmText:='File Delete Error While Deleting Old Log',sRcyText:='An Error Was Encountered While Trying To Delete File. Please Contact Nutek For A Possible Solution.'),(sAlmText:='Receive Check Alive While In Remote Configuration',sRcyText:='Receive Illegal Message.'),(sAlmText:='Receive Check Alive Ping While In Remote Configuration',sRcyText:='Receive Illegal Message.'),(sAlmText:='Receive Check Alive Pong While In Remote Configuration',sRcyText:='Receive Illegal Message.'),(sAlmText:='Receive ServiceDescription While In Remote Configuration',sRcyText:='Receive Illegal Message.'),(sAlmText:='Receive BoardAvailable While In Remote Configuration',sRcyText:='Receive Illegal Message.'),(sAlmText:='Receive RevokeBoardAvailable While In Remote Configuration',sRcyText:='Receive Illegal Message.'),(sAlmText:='Receive MachineReady While In Remote Configuration',sRcyText:='Receive Illegal Message.'),(sAlmText:='Receive RevokeMachineReady While In Remote Configuration',sRcyText:='Receive Illegal Message.'),(sAlmText:='Receive StartTransport While In Remote Configuration',sRcyText:='Receive Illegal Message.'),(sAlmText:='Receive StopTransport While In Remote Configuration',sRcyText:='Receive Illegal Message.'),(sAlmText:='Receive TransportFinished While In Remote Configuration',sRcyText:='Receive Illegal Message.'),(sAlmText:='Receive CurrentConfiguration While In Remote Configuration',sRcyText:='Receive Illegal Message.'),(sAlmText:='Receive BoardForecast While In Remote Configuration',sRcyText:='Receive Illegal Message.'),(sAlmText:='Receive QueryBoardInfo While In Remote Configuration',sRcyText:='Receive Illegal Message.'),(sAlmText:='Receive SendBoardInfo While In Remote Configuration',sRcyText:='Receive Illegal Message.'),(sRcyText:='Sending Illegal Message.'),(sAlmText:='Service Description Request To Send From Remote Hermes',sRcyText:='Sending Illegal Message.'),(sAlmText:='Board Available Request To Send From Remote Hermes',sRcyText:='Sending Illegal Message.'),(sAlmText:='Revoke Board Available Request To Send From Remote Hermes',sRcyText:='Sending Illegal Message.'),(sAlmText:='Stop Transport Request To Send From Remote Hermes',sRcyText:='Sending Illegal Message.'),(sAlmText:='Transport Finished Request To Send From Remote Hermes',sRcyText:='Sending Illegal Message.'),(sAlmText:='Machine Ready Request To Send From Remote Hermes',sRcyText:='Sending Illegal Message.'),(sAlmText:='Revoke Machine Ready Request To Send From Remote Hermes',sRcyText:='Sending Illegal Message.'),(sAlmText:='Start Transport Request To Send From Remote Hermes',sRcyText:='Sending Illegal Message.'),(sAlmText:='Set Configuration Request To Send From Remote Hermes',sRcyText:='Sending Illegal Message.'),(sAlmText:='Get Configuration Request To Send From Remote Hermes',sRcyText:='Sending Illegal Message.'),(sAlmText:='Current Configuration Request To Send From Remote Hermes',sRcyText:='Sending Illegal Message.'),(sAlmText:='Board Forecast Request To Send From Remote Hermes',sRcyText:='Sending Illegal Message.'),(sAlmText:='Query Board Info Request To Send From Remote Hermes',sRcyText:='Sending Illegal Message.'),(sAlmText:='Invalid Ident While Sending Data',sRcyText:='Invalid Ident Value.'),(sAlmText:='TCP Retry Send Data Error While Sending Data',sRcyText:='Problem Occurred In The TCP/IP Connection. Check The Connection And Try To Reconnect.'),(sAlmText:='TCP Send Data Error',sRcyText:='Problem Occurred In The TCP/IP Connection. Check The Connection And Try To Reconnect.'),(sAlmText:='Invalid Ident While Closing TCP',sRcyText:='Invalid Ident Value.'),(sAlmText:='Closing TCP Error',sRcyText:='Problem Occurred In The TCP/IP Connection. Check The Connection And Try To Reconnect.'),(sAlmText:='File Open Error While Writing Log',sRcyText:='An Error Was Encountered While Trying To Open File. Please Contact Nutek For A Possible Solution.'),(sAlmText:='File Create Error While Writing Log',sRcyText:='An Error Was Encountered While Trying To Create File. Please Contact Nutek For A Possible Solution.'),(sAlmText:='Get File Info Error While Writing Log',sRcyText:='An Error Was Encountered While Getting File Info. Please Contact Nutek For A Possible Solution.'),(sAlmText:='File Write Error While Writing Log',sRcyText:='An Error Was Encountered While Trying To Write File. Please Contact Nutek For A Possible Solution.'),(sAlmText:='File Close Error While Writing Log',sRcyText:='An Error Was Encountered While Trying To Close File. Please Contact Nutek For A Possible Solution.'),(sAlmText:='Directory Does Not Exist While Writing Log',sRcyText:='The Directory Does Not Exist.Please Contact Nutek For A Possible Solution.'),(sAlmText:='Invalid Ident While Closing TCP',sRcyText:='Invalid Ident Value.'),(sAlmText:='Closing TCP Error',sRcyText:='Problem Occurred In The TCP/IP Connection. Check The Connection And Try To Reconnect.'),3((0)),(sAlmText:='Send Board Info Request To Send From Upstream Hermes',sRcyText:='Sending Illegal Message.'),(sAlmText:='Query Work Order Info Request To Send From Upstream Hermes',sRcyText:='Sending Illegal Message.'),(sAlmText:='Send Work Order Info Request To Send From Upstream Hermes',sRcyText:='Sending Illegal Message.'),(sAlmText:='Board Arrived Request To Send From Upstream Hermes',sRcyText:='Sending Illegal Message.'),(sAlmText:='Board Departed Request To Send From Upstream Hermes',sRcyText:='Sending Illegal Message.'),36((0))];
END_VAR
(**)
(*Local Output*)
VAR
	bFileNotFound : BOOL;
	bConnected : BOOL;
	bWriteConfig : BOOL := FALSE;
	bUpdateUIData : BOOL := FALSE;
	tyCurrentConfiguration : tyHermesCurrentConfiguration;
END_VAR
(**)
(*Local Input*)
VAR
	udiRstErr : UDINT := 0;
	bPrep : BOOL := TRUE;
	bEn : BOOL := TRUE;
	bDis : BOOL := FALSE;
	bRmtPrep : BOOL := FALSE;
	bRmtEn : BOOL := FALSE;
	tyParam : tyHermesRmtParam := (uiSvrPort:=1248);
	sIPAddr : STRING[15] := '192.168.0.100';
	tyDTStructure : DTStructure := (year:=2020,month:=11,day:=11,wday:=05,hour:=21,minute:=28,second:=30,millisec:=123,microsec:=456);
	dtCurrDT : DATE_AND_TIME := DT#2019-02-23-12:30:50;
	sMcId : STRING[80] := '';
	udiSndBffrSize : UDINT := 65536;
	udiRcvBffrSize : UDINT := 65536;
	udiAliveIdleTimeInSec : UDINT := 5;
	udiFileKeepDay : UDINT := 30;
	sConfigFileName : STRING[80] := 'RmtHermes.dat';
	sProgNm : STRING[15] := 'RmtHermes';
	bNtSettingsLoadDone : BOOL := TRUE;
	tyHermesCurrConfiguration : tyHermesConfiguration;
END_VAR
(**)
(*Local*)
VAR
	bRstErr : BOOL;
	udiRstErrOld : UDINT;
	bInitDone : BOOL;
	bInitialDone : BOOL;
	bRun : BOOL;
	bStop : BOOL;
	bRstConnection : BOOL;
	udiSvrIdent : UDINT;
	udiClntIdent : UDINT;
	udiXMLTableWriteIdx : UDINT;
	udiMsgSendBffr : UDINT;
	udiSndMsgLen : UDINT;
	sSnd : STRING[65535];
	sRcv : STRING[65535];
	a_tyXMLTableDataRcv : ARRAY[0..200] OF tyXMLTableDat;
	a_tyXMLTableDataSnd : ARRAY[0..200] OF tyXMLTableDat;
	a_eMsgSend : ARRAY[0..50] OF eHermesMsgType;
	tyMsgTypeRcv : tyHermesMsgType;
	tyCheckAlive : tyHermesCheckAlive;
	tyCheckAlivePing : tyHermesCheckAlive;
	tyCheckAlivePong : tyHermesCheckAlive;
	tyServiceDescriptionRcv : tyHermesServiceDescription;
	tyNotificationSnd : tyHermesNotification;
	tyNotificationRcv : tyHermesNotification;
	tyBoardAvailableRcv : tyHermesBoardAvailable;
	tyMachineReady : tyHermesMachineReady;
	tyStartTransport : tyHermesStartTransport;
	tyStopTransport : tyHermesStopTransport;
	tyTransportFinished : tyHermesTransportFinished;
	tySetConfiguration : tyHermesSetConfiguration;
	tySetConfigurationRcv : tyHermesSetConfiguration;
	tySetConfigurationModified : tyHermesSetConfiguration;
	tyCurrentConfigurationRcv : tyHermesCurrentConfiguration;
	tyCurrentConfigurationSnd : tyHermesCurrentConfiguration;
	tyBoardForecast : tyHermesBoardForecast;
	tyQueryBoardInfo : tyHermesQueryBoardInfo;
	tySendBoardInfo : tyHermesSendBoardInfo;
	fbCreateSvr : fbTCPCreateSvr;
	fbListen : fbTCPListen;
	fbRcv : fbTCPRcv;
	fbSend : fbTCPSnd;
	fbCloseSvr : fbTCPClose;
	fbCloseClnt : fbTCPClose;
	fbParseXMLTable : fbHermesParseXMLTable;
	eStatOld : eHermesAction := HermesActIdle;
	tyParamOld : tyHermesRmtParam;
	udiLogCntr : UDINT := 1;
	udiWriteLogCntr : UDINT := 1;
	a_sLogList : ARRAY[1..10] OF STRING[65535];
	sDT : STRING[80];
	dtCurrDTTemp : DATE_AND_TIME;
	fbFileAppend1 : fbFileFullAppend;
	fbFileOldDel1 : fbFileOldDel;
	fbDelayTm : TON;
	fbDelayTm1 : TON;
	bFoundIndexUS1 : BOOL;
	bFoundIndexUS2 : BOOL;
	bFoundIndexUS3 : BOOL;
	bFoundIndexUS4 : BOOL;
	bFoundIndexDS1 : BOOL;
	bFoundIndexDS2 : BOOL;
	bFoundIndexDS3 : BOOL;
	bFoundIndexDS4 : BOOL;
	udiFoundIndexUS1 : UDINT;
	udiFoundIndexUS2 : UDINT;
	udiFoundIndexUS3 : UDINT;
	udiFoundIndexUS4 : UDINT;
	udiFoundIndexDS1 : UDINT;
	udiFoundIndexDS2 : UDINT;
	udiFoundIndexDS3 : UDINT;
	udiFoundIndexDS4 : UDINT;
	udiTargetAddress : UDINT := 0;
	udiTargetAddress1 : UDINT := 0;
	udiSizeAddress : UDINT := 0;
	udiSizeAddress1 : UDINT := 0;
	k : UDINT := 0;
	kk : UDINT := 0;
	j : INT := 1;
	jj : INT := 2;
	jjj : INT := 3;
	jjjj : INT := 4;
	i : INT;
	ii : INT;
	iii : INT;
	iiii : INT;
	iInput : INT := 1;
	iOutput : INT := 1;
	iWriteLogStep : INT := 0;
	udiModuleNum : UDINT := 3601;
END_VAR
```

### SvyHermes.var - Change By Project
```iecst
(*2021-08-01*)
(**)
(*Action & State & Status*)
VAR
	p_SvyHermesStat : UDINT;
	p_SvyHermesStatus : UDINT;
	p_SvyHermesStatTxt : UDINT;
	p_SvyHermesAct : UDINT;
	p_SvyHermesMcParamAct : UDINT;
END_VAR
(**)
(*Alarm*)
VAR
	p_SvyHermesAlmData : UDINT;
	p_SvyHermesAlmData1 : UDINT;
	p_SvyHermesAlmData2 : UDINT;
	p_SvyHermesAlmData3 : UDINT;
	p_SvyHermesAlmData4 : UDINT;
	p_SvyHermesInfoData : UDINT;
	p_SvyHermesInfoData1 : UDINT;
	p_SvyHermesInfoData2 : UDINT;
	p_SvyHermesInfoData3 : UDINT;
	p_SvyHermesInfoData4 : UDINT;
	p_SvyHermesInfoData5 : UDINT;
	p_SvyHermesInfoData6 : UDINT;
END_VAR
(**)
(*Output*)
VAR
	p_SvyHermesConnected : UDINT;
	p_SvyHermesHandshakeDone : UDINT;
	p_SvyHermesFileNotFound : UDINT;
	p_SvyHermesSetConfiguration : UDINT;
	p_SvyHermesWriteConfig : UDINT;
	p_SvyHermesUpdateUIData : UDINT;
	p_SvyHermesInternalSnd : UDINT;
	p_SvyHermesWorkOrderId : UDINT;
	p_SvyHermesBatchId : UDINT;
	p_SvyHermesFoundIndexUS1 : UDINT;
	p_SvyHermesFoundIndexUS2 : UDINT;
	p_SvyHermesFoundIndexUS3 : UDINT;
	p_SvyHermesFoundIndexUS4 : UDINT;
	p_SvyHermesFoundIndexDS1 : UDINT;
	p_SvyHermesFoundIndexDS2 : UDINT;
	p_SvyHermesFoundIndexDS3 : UDINT;
	p_SvyHermesFoundIndexDS4 : UDINT;
	p_SvyHermesIndexUS1 : UDINT;
	p_SvyHermesIndexUS2 : UDINT;
	p_SvyHermesIndexUS3 : UDINT;
	p_SvyHermesIndexUS4 : UDINT;
	p_SvyHermesIndexDS1 : UDINT;
	p_SvyHermesIndexDS2 : UDINT;
	p_SvyHermesIndexDS3 : UDINT;
	p_SvyHermesIndexDS4 : UDINT;
	p_SvyHermesSendWorkOrderInfo : UDINT;
	p_SvyHermesRcvInsertBoardInfo : UDINT;
	p_RcvWorkOrderInfo1 : UDINT;
	p_ManualInsertData : UDINT := 0;
END_VAR
```

### Program Logical/Hermes/SvyHermes (IEC, version 1.00.0) - 1.00.1 - NtHermes v5.00.4 , NtTCP v5.00.2 , NtMessage v5.00.1

#### Init.st - Change By Project
```iecst
(** 2021-08-01 **)
PROGRAM _INIT

	(* Always Change If Project Change *)

	//Pass Address To Global Address For External Use
	//Action, State & Status
	p_SvyHermesStat	    	:= ADR(eStat);
	p_SvyHermesStatus   	:= ADR(eMainStatus);
	p_SvyHermesStatTxt    	:= ADR(sStatTxt);
	p_SvyHermesAct	    	:= ADR(eHermesAct);
	p_SvyHermesMcParamAct	:= ADR(eMcParamAct);

	//Alarm
	p_SvyHermesAlmData	    := ADR(tyAlmData);
	p_SvyHermesAlmData1	    := ADR(tyAlmData1);
	p_SvyHermesAlmData2	    := ADR(tyAlmData2);
	p_SvyHermesAlmData3	    := ADR(tyAlmData3);
    p_SvyHermesAlmData4	    := ADR(tyAlmData4);
	p_SvyHermesInfoData	    := ADR(tyInfoData);
	p_SvyHermesInfoData1	:= ADR(tyInfoData1);
	p_SvyHermesInfoData2	:= ADR(tyInfoData2);
	p_SvyHermesInfoData3	:= ADR(tyInfoData3);
	p_SvyHermesInfoData4	:= ADR(tyInfoData4);
	p_SvyHermesInfoData5	:= ADR(tyInfoData5);
	p_SvyHermesInfoData6	:= ADR(tyInfoData6);

	//Output
	p_SvyHermesConnected			:= ADR(bConnected);
	p_SvyHermesHandshakeDone		:= ADR(bHandshakeDone);
	p_SvyHermesInternalSnd		    := ADR(sInternalSnd);
	p_SvyHermesFileNotFound			:= ADR(bFileNotFound);
	p_SvyHermesSetConfiguration	    := ADR(tySetConfigurationModified);
	p_SvyHermesWriteConfig	        := ADR(bWriteConfig);
	p_SvyHermesUpdateUIData	        := ADR(bUpdateUIData);
	p_SvyHermesWorkOrderId          := ADR(sWorkOrderId); //WorkOrderId from Supervisory System
	p_SvyHermesBatchId              := ADR(sBatchId); //BatchId from Supervisory System
	p_SvyHermesSendWorkOrderInfo    := ADR (tySendWorkOrderInfoRcv);   // Pass Receive data to Downstream
	p_SvyHermesRcvInsertBoardInfo	:= ADR(bRcvInsertBoardInfo);

	//Data
	p_SvyHermesFoundIndexUS1              := ADR(bFoundIndexUS1);
	p_SvyHermesFoundIndexUS2              := ADR(bFoundIndexUS2);
	p_SvyHermesFoundIndexUS3              := ADR(bFoundIndexUS3);
	p_SvyHermesFoundIndexUS4              := ADR(bFoundIndexUS4);
	p_SvyHermesFoundIndexDS1              := ADR(bFoundIndexDS1);
	p_SvyHermesFoundIndexDS2              := ADR(bFoundIndexDS2);
	p_SvyHermesFoundIndexDS3              := ADR(bFoundIndexDS3);
	p_SvyHermesFoundIndexDS4              := ADR(bFoundIndexDS4);
	p_SvyHermesIndexUS1                   := ADR(udiFoundIndexUS1);
	p_SvyHermesIndexUS2                   := ADR(udiFoundIndexUS2);
	p_SvyHermesIndexUS3                   := ADR(udiFoundIndexUS3);
	p_SvyHermesIndexUS4                   := ADR(udiFoundIndexUS4);
	p_SvyHermesIndexDS1                   := ADR(udiFoundIndexDS1);
	p_SvyHermesIndexDS2                   := ADR(udiFoundIndexDS2);
	p_SvyHermesIndexDS3                   := ADR(udiFoundIndexDS3);
	p_SvyHermesIndexDS4                   := ADR(udiFoundIndexDS4);

	//Add
	p_RcvWorkOrderInfo1                := ADR(bRcvWorkOrderInfo1);
	p_ManualInsertData                 := ADR(bManualInsertData);

	(* Always Change If Project Change *)

END_PROGRAM
```

#### Act_InitGlobal.st - Change By Project
```iecst
(** 2021-08-01 **)
ACTION Act_InitGlobal:

	(* Always Change If Project Change *)

	//Pass Data To Link
	p_bLinkStartupRun ACCESS p_StartupRun;

	//Pass Data To Internal Use
	p_udiRstErr ACCESS p_RstErrReset;
	p_bPrep ACCESS p_NtParamHermesPrep;
	p_tyParam ACCESS p_HermesSvyParam;
	p_sIPAddr ACCESS p_HWInfoIPAddr;
	pa_usiMacAddr ACCESS p_HWInfoMacAddr;
	p_tyDTStructure ACCESS p_TimeCurrDTStruct;
	p_dtCurrDT ACCESS p_TimeCurrDT;
	p_sMcId ACCESS p_McParamMcNm;
	p_sRecipeNm ACCESS p_ProdRcpCurrRcp0Nm;
	p_sMagazineId ACCESS p_UIMagazineId;
	p_iSlotId ACCESS p_UIMagazineSlotId;
	p_sBarcode ACCESS p_UIPCBBarcode;
	p_udiAliveIdleTimeInSec ACCESS p_NtParamSvyHermesAliveTmInSec;
	p_tConnTimeOut ACCESS p_NtParamSvyHermesConnTO;
	p_diTransferInTO ACCESS p_McParamTranOutErrDlyTm;
	p_bNewBrdAvlLastZone ACCESS p_HermesBrdAvlDataNewBrdAvlLastZ;
	p_bOpsRun ACCESS p_OpsRun;
	p_udiFileKeepDay ACCESS p_NtParamSvyHermesFileKeepDay;
	p_sConfigFileName ACCESS p_NtParamSvyHermesConfigFileNm;
	p_sProgNm ACCESS p_NtParamSvyHermesProgNm;
	p_bNtSettingsLoadDone ACCESS p_StartupNtSettingsLoadDone;
	p_bSvyPrep ACCESS p_NtParamHermesSvyPrep;
	p_bSvyEn ACCESS p_McParamHermesSvyEn;
	p_bQueryWorkOrderInfo ACCESS p_UIQueryWorkOrderInfo;
	p_bReinsertBrd ACCESS p_UIReinsertBrd;
	p_bInsertBoard ACCESS p_UIInsertBoard;
	p_tyHermesConfiguration ACCESS p_HermesConfiguration;
	p_bUSHermesStopTransport1 ACCESS p_USHermesStopTransportSnd; //Lane 1
//	p_bUSHermesStopTransport2 ACCESS p_USHermesStopTransportSnd2; //Lane 2, open up for specific machine
//	p_bUSHermesStopTransport3 ACCESS p_USHermesStopTransportSnd3; //Lane 3, open up for specific machine
//	p_bUSHermesStopTransport4 ACCESS p_USHermesStopTransportSnd4; //Lane 4, open up for specific machine
	p_tyUSBoardArrived1 ACCESS p_USHermesBoardArrivedData; //Lane 1
//	p_tyUSBoardArrived2 ACCESS p_USHermesBoardArrivedData2; //Lane 2, open up for specific machine
//	p_tyUSBoardArrived3 ACCESS p_USHermesBoardArrivedData3; //Lane 3, open up for specific machine
//	p_tyUSBoardArrived4 ACCESS p_USHermesBoardArrivedData4; //Lane 4, open up for specific machine
	p_bDSHermesTransportFinished1 ACCESS p_DSHermesTransportFinishedSnd;
//	p_bDSHermesTransportFinished2 ACCESS p_DSHermesTransportFinishedSnd2; //Lane 2, open up for specific machine
//	p_bDSHermesTransportFinished3 ACCESS p_DSHermesTransportFinishedSnd3; //Lane 3, open up for specific machine
//	p_bDSHermesTransportFinished4 ACCESS p_DSHermesTransportFinishedSnd4; //Lane 4, open up for specific machine
	p_tyDSBoardDeparted1 ACCESS p_DSHermesBoardDepartedData; //Lane 1
//	p_tyDSBoardDeparted2 ACCESS p_DSHermesBoardDepartedData2; //Lane 2, open up for specific machine
//	p_tyDSBoardDeparted3 ACCESS p_DSHermesBoardDepartedData3; //Lane 3, open up for specific machine
//	p_tyDSBoardDeparted4 ACCESS p_DSHermesBoardDepartedData4; //Lane 4, open up for specific machine
	p_eHermesStat ACCESS p_HermesStat;
	p_eHermesStatus ACCESS p_HermesStatus;
	p_eMcParamStat ACCESS p_McParamStat;
	p_eMcParamStatus ACCESS p_McParamStatus;
	p_bAllZonesEmpty ACCESS p_DSHermesAllZonesEmpty; //All zones empty. Before empty, cannot change current sWorkOrderId.
	p_bDeleteWorkOrder ACCESS p_UIDeleteWorkOrder;
	p_bFirstMcIntheLine ACCESS p_NtParamHermesSvyFirstMc; //First machine in the line only can Query Work Order
	p_sRetainFileName ACCESS p_NtParamSvyHermesRetainFileNm;
	p_bHermesSvyQueryBoardInfo ACCESS p_NtParamHermesSvyQueryBoardInfo;
	p_bHermesReinsertBoard ACCESS p_NtParamHermesReinsertBoard;
	p_bConvRgtSen ACCESS p_DIConvRgtSen;
	p_bConvLftSen ACCESS p_DIConvLftSen;
	p_tyProdRcpCurrRcp ACCESS p_ProdRcpCurrRcp0;
	p_tyMcParamCurr	ACCESS p_McParamCurr;
	p_tyNtParamCurr	ACCESS p_NtParamCurr;
	p_eLinkMcParamDSCommMod ACCESS p_McParamDSCommMod;
	p_bAWWidthPosDiff ACCESS p_AWOpenWidthPosDiff;           //Add
	p_bOpsGConvStepEntBrd ACCESS p_OpsGConvStepEntBrd;
	p_bOpsGConvStepDSTmr ACCESS p_OpsGConvStepDSTmr;
	p_bOpsGConvStepDSCommTmr ACCESS p_OpsGConvStepDSCommTmr;

	//	p_bRemovedBoard ACCESS p_RemovedBoard;               //ADD
	(* Always Change If Project Change *)
END_ACTION
```

#### InputRef_Link.var - Change By Project
```iecst
(*2021-08-01*)
(**)
VAR
	p_bLinkStartupRun : REFERENCE TO BOOL;
	bHermesRun : BOOL;
	bHermesStop : BOOL;
END_VAR
(**)
```

#### Act_LinkAction.st - Change By Project
```iecst
(** 2021-08-01 **)
ACTION Act_LinkAction:

	IF p_bLinkStartupRun = TRUE THEN
		p_eAct ACCESS p_StartupSvyHermesAct;
	ELSE
		p_eAct ACCESS ADR(eAct);

		IF EDGEPOS(p_bSvyPrep AND p_bSvyEn) THEN
			bHermesRun	:= TRUE;
			bHermesStop	:= FALSE;
		END_IF

		IF EDGENEG(p_bSvyPrep AND p_bSvyEn) THEN
			bHermesRun	:= FALSE;
			bHermesStop	:= TRUE;
		END_IF

		IF bHermesRun = TRUE THEN
			p_eAct	:= HermesActBGStartRun;

			IF (eStat = HermesActBGStartRun) AND (eStatus = Done) THEN
				p_eAct			:= HermesActIdle;
				bHermesRun	:= FALSE;
			END_IF
		END_IF

		IF bHermesStop = TRUE THEN
			p_eAct	:= HermesActBGStopRun;

			IF (eStat = HermesActBGStopRun) AND (eStatus = Done) THEN
				p_eAct	    := HermesActIdle;
				bHermesStop	:= FALSE;
			END_IF
		END_IF

	END_IF

END_ACTION
```

#### Act_Link.st - Change By Project
```iecst
(** 2021-08-01 **)
ACTION Act_Link:

	//Receive Alive Time
	p_tyParam.tRcvAlive	:= p_tyParam.tSndAlive * 2;

	// For BoardDeparted's BoardTransfer Parameter
	IF p_bFirstMcIntheLine = TRUE AND p_bNewBrdAvlLastZone THEN
		p_eBoardTransfer1 := HermesInserted;
	ELSIF p_bFirstMcIntheLine = TRUE AND p_bNewBrdAvlLastZone = FALSE THEN
		p_eBoardTransfer1 := HermesTransferred;
	ELSIF p_bFirstMcIntheLine = FALSE AND p_bNewBrdAvlLastZone THEN
		p_eBoardTransfer1 := HermesInserted;
	ELSIF p_bFirstMcIntheLine = FALSE AND p_bNewBrdAvlLastZone = FALSE THEN
		p_eBoardTransfer1 := HermesTransferred;
	END_IF

	//Info Message
	p_sInfoMsg		:= 'Hermes Configuration Received From Supervisory System';

	//Info Message 1
	p_sInfoMsg1     := 'Work Order Info Received From Supervisory System';
	p_sInfoMsg1		:= CONCAT(p_sInfoMsg1 , '$r$n');
	p_sInfoMsg1		:= CONCAT(p_sInfoMsg1 , 'PCB Work Order Info Will Be Overwritten');

	//Info Message 2
	p_sInfoMsg2     := 'Work Order Info Not Found From Supervisory System';
	p_sInfoMsg2		:= CONCAT(p_sInfoMsg2 , '$r$n');
	p_sInfoMsg2  	:= CONCAT(p_sInfoMsg2 , 'Please Try Again');

	//Info Message 3
	p_sInfoMsg3     := 'Query Work Order Not Possible';
	p_sInfoMsg3		:= CONCAT(p_sInfoMsg3 , '$r$n');
	p_sInfoMsg3  	:= CONCAT(p_sInfoMsg3 , 'Please Empty the Machines');
	p_sInfoMsg3		:= CONCAT(p_sInfoMsg3 , '$r$n');
	p_sInfoMsg3  	:= CONCAT(p_sInfoMsg3 , 'and Try Again');

	//Info Message 4
	p_sInfoMsg4     := 'Waiting For LCS';

	//Info Message 5
	p_sInfoMsg5     := 'Waiting for Board insert';

	//Info Message 6
	p_sInfoMsg6     := 'Remove Board';

	//Accept WorkOrderId from Supervisory System, adjust accordingly
	//(Loader Machine: Magazine area empty, Lifter area empty)
	//(Destacker Machine: load pcb stack area empty and conveyor empty)
	p_bAcceptCondition := p_bAllZonesEmpty;

END_ACTION
```

#### Cyclic.st - Do Not Change!!!
```iecst
(** 2021-08-01 **)
PROGRAM _CYCLIC

	IF bInitDone = FALSE THEN
		bInitDone	:= TRUE;

		Act_InitLocal;
		Act_InitGlobal;

	ELSIF bInitialDone = FALSE THEN
		IF p_bNtSettingsLoadDone = TRUE THEN
			bInitialDone	:= TRUE;

			Act_Initial;
		END_IF

	ELSE

		Act_RstErr;
		Act_LinkAction;
		Act_Action;
		Act_LinkEn;

		IF (p_bPrep = TRUE) AND (p_bEn = TRUE) AND (p_bDis = FALSE) THEN
			Act_Link;
			Act_Main;
			Act_Background;
			Act_Background_ProcessData;
		ELSE
			Act_Main_Disable;

			IF eStat <> HermesActIdle THEN
				eStatus	:= Done;
			ELSE
				eStatus	:= Idle;
			END_IF
		END_IF

		Act_CombineErr;
		Act_Alarm;
		Act_Alarm1;
		Act_Alarm2;
		Act_Alarm3;
		Act_Alarm4;

	END_IF

END_PROGRAM
```
